// TwinCAT 3 PLC project Plc1
// ProgramVersion: 3.1.4023.0
// libraries:
//   Tc2_Standard, * (Beckhoff Automation GmbH)
//   Tc2_System, * (Beckhoff Automation GmbH)
//   Tc3_Module, * (Beckhoff Automation GmbH)
//   TcoCore, 0.9.0.4 (Vortex.Library)
//   TcoIo, 0.9.0.4 (Vortex.Library)
// project tree:
//   / PlcTask.TcTTO
//   POUs/ MAIN.TcPOU
//   DUTs/IO/PdoEntries/ Status_3D84275F.TcDUT, Ctrl_1EFB4D3B.TcDUT, Ctrl_71604E86.TcDUT, Status_B0753356.TcDUT, Status_F2CE6D91.TcDUT, U1_Status_DC903920.TcDUT, U1_Samples_25492287.TcDUT, I1_Status_DC903920.TcDUT, I1_Samples_25492287.TcDUT, U2_Status_DC903920.TcDUT, U2_Samples_25492287.TcDUT, I2_Status_DC903920.TcDUT, I2_Samples_25492287.TcDUT, U3_Status_DC903920.TcDUT, U3_Samples_25492287.TcDUT, I3_Status_DC903920.TcDUT, I3_Samples_25492287.TcDUT, StartTimeNextLatch_02E0C1C8.TcDUT, Status_642C2ED1.TcDUT, Ctrl_77460BD3.TcDUT, Outputs_A910484D.TcDUT
//   DUTs/IO/PDOs/ COM_TxPDO_Map_Inputs_Channel_3801C95E.TcDUT, COM_RxPDO_Map_Outputs_Channel_EADA2E0D.TcDUT, Channel_830843C1.TcDUT, Channel_42CA91F7.TcDUT, AO_Output_Channel_BA7EBB7C.TcDUT, COM_Inputs_3801C95E.TcDUT, COM_Outputs_DEF408EC.TcDUT, AI_Standard_Channel_A8DF64E3.TcDUT, AI_Standard_Channel_4A394481.TcDUT, L1_Voltage_Status_7371B043.TcDUT, L1_Voltage_Samples_41AEB7FF.TcDUT, L1_Current_Status_82DECBF6.TcDUT, L1_Current_Samples_9EC08B3E.TcDUT, L2_Voltage_Status_0D1813FE.TcDUT, L2_Voltage_Samples_75D833AF.TcDUT, L2_Current_Status_FCB7684B.TcDUT, L2_Current_Samples_AAB60F6E.TcDUT, L3_Voltage_Status_273F7295.TcDUT, L3_Voltage_Samples_660A4F9F.TcDUT, L3_Current_Status_D6900920.TcDUT, L3_Current_Samples_B964735E.TcDUT, AI_NextSync1Time_6DC4D296.TcDUT, AI_Sample_Count_EA88CAD9.TcDUT, InfoData_B84DBEC5.TcDUT, MTO_Inputs_Channel_53C09E8B.TcDUT, MTO_Outputs_10x_Channel_A3C0C022.TcDUT, PM_Inputs_Channel_2F868086.TcDUT, PM_Status_data_2A9514CB.TcDUT, PM_Outputs_Channel_E5FBDE30.TcDUT, AT_x_4EC2E768.TcDUT, MDT_864618EC.TcDUT, InfoData_F60A43AC.TcDUT
//   DUTs/IO/Boxes/ EK1200_013D0B49.TcDUT, EL6002_CD897635.TcDUT, EL1809_32157CFD.TcDUT, EL2809_2B6483BD.TcDUT, EL4004_E203F875.TcDUT, EL6001_0DE01E7E.TcDUT, EL9011_D65D3D32.TcDUT, EK1100_1FC0878B.TcDUT, EK1122_1FC0878B.TcDUT, EL3174_B71BFF42.TcDUT, EL3011_7A495228.TcDUT, EL2008_E2806B95.TcDUT, EK1110_1FC0878B.TcDUT, EL1819_32157CFD.TcDUT, EL2788_E2806B95.TcDUT, EL3773_F128CC82.TcDUT, EL2258_E3B260FA.TcDUT, EL3164_B71BFF42.TcDUT, EL1008_78E8D3DD.TcDUT, EL3403_812980A6.TcDUT, EL3024_C6E76B5A.TcDUT, AX5101_1BD22F51.TcDUT
//   DUTs/IO/Devices/ SyncUnitTasks_4BE01469.TcDUT, SyncUnits_67D36DDA.TcDUT, SyncUnits_91A42BBF.TcDUT
//   DUTs/IO/Topology/ Term_1_EK1200_B38DC9A8.TcDUT, Device_1_EtherCAT_B557D6C6.TcDUT, Term_11_EK1100_B6553301.TcDUT, Term_18_EK1100_20659A8D.TcDUT, Term_25_EK1100_08217EB4.TcDUT, Term_28_EK1100_415F4A7E.TcDUT, Term_24_EK1122_39E7B5CB.TcDUT, Term_23_EK1100_C1096874.TcDUT, Term_42_EK1100_1039F2C4.TcDUT, Term_10_EK1122_152EB6C2.TcDUT, Term_9_EK1100_0DC40061.TcDUT, Device_2_EtherCAT_CA128DDC.TcDUT, Term_157_EK1100_7C4BDD77.TcDUT, Term_158_EK1100_E3D699B1.TcDUT, Term_154_EK1122_E57516AE.TcDUT, Term_153_EK1100_91C0BB48.TcDUT, Term_180_EK1100_796B7783.TcDUT, Term_182_EK1100_E6B2C35E.TcDUT, Term_179_EK1122_2A33725A.TcDUT, Term_178_EK1100_9B7E9852.TcDUT, Term_147_EK1122_CA6A5D16.TcDUT, Term_189_EK1100_06A16014.TcDUT, Term_194_EK1100_D4E2C05F.TcDUT, Term_188_EK1122_78D8AA43.TcDUT, Term_187_EK1100_648C31BD.TcDUT, Term_231_EK1100_6FCE8CEB.TcDUT, Term_233_EK1100_CB654C3B.TcDUT, Term_230_EK1122_16418046.TcDUT, Term_207_EK1100_2D36550A.TcDUT, Term_186_EK1122_75C79D52.TcDUT, Term_237_EK1122_86A8F7BD.TcDUT, Term_289_EK1100_9C677E50.TcDUT, Term_294_EK1100_DFE2A59E.TcDUT, Term_331_EK1100_B9C4E092.TcDUT, Term_333_EK1100_1D6F2042.TcDUT, Term_330_EK1122_0EDE60FE.TcDUT, Term_307_EK1100_EB8FAA41.TcDUT, Term_288_EK1122_18F8921F.TcDUT, Term_146_EK1100_439F5464.TcDUT, Device_3_EtherCAT_CA191EDE.TcDUT
//   GVLs/ GVL_iXlinker.TcGVL
// real-time tasks:
//   TASK PlcTask: cycle T#10ms, priority 20, ADS port 350
// I/O:
//   DEVICE Device 1 (EtherCAT) (disabled), AmsNetId 172.20.10.110.2.1
//     Term 1 (EK1200) [EK1200-5000 EtherCAT Power supply (2A E-Bus)]
//       Term 2 (EL6002) [EL6002 Interface 2Ch. (RS232)]
//       Term 3 (EL1809) [EL1809 16Ch. Dig. Input 24V, 3ms]
//       Term 4 (EL2809) [EL2809 16Ch. Dig. Output 24V, 0.5A]
//       Term 5 (EL4004) [EL4004 4Ch. Ana. Output 0-10V, 12bit]
//       Term 6 (EL2809) [EL2809 16Ch. Dig. Output 24V, 0.5A]
//       Term 7 (EL6001) [EL6001 Interface (RS232)]
//       Term 8 (EL9011) [EL9011 End Terminal]
//   DEVICE Device 2 (EtherCAT) (disabled), AmsNetId 172.20.10.110.3.1
//     Term 9 (EK1100) [EK1100 EtherCAT Coupler (2A E-Bus)]
//       Term 10 (EK1122) [EK1122 2 port EtherCAT junction]
//         Term 11 (EK1100) [EK1100 EtherCAT Coupler (2A E-Bus)]
//           Term 12 (EL3174-0002) [EL3174-0002 4Ch. Ana. Input +/-10V, +/-20mA 16 Bit, Isolated Channels]
//           Term 13 (EL6001) [EL6001 Interface (RS232)]
//           Term 14 (EL3011) [EL3011 4Ch. Ana. Input 0-20mA DIFF]
//           Term 15 (EL2008) [EL2008 8Ch. Dig. Output 24V, 0.5A]
//           Term 16 (EL2008) [EL2008 8Ch. Dig. Output 24V, 0.5A]
//           Term 17 (EK1110) [EK1110 EtherCAT extension]
//         Term 18 (EK1100) [EK1100 EtherCAT Coupler (2A E-Bus)]
//           Term 19 (EL1809) [EL1809 16Ch. Dig. Input 24V, 3ms]
//           Term 20 (EL2809) [EL2809 16Ch. Dig. Output 24V, 0.5A]
//           Term 21 (EL1809) [EL1809 16Ch. Dig. Input 24V, 3ms]
//           Term 22 (EL3011) [EL3011 4Ch. Ana. Input 0-20mA DIFF]
//           Term 29 (EL9011) [EL9011 End Terminal]
//         Term 23 (EK1100) [EK1100 EtherCAT Coupler (2A E-Bus)]
//           Term 24 (EK1122) [EK1122 2 port EtherCAT junction]
//             Term 25 (EK1100) [EK1100 EtherCAT Coupler (2A E-Bus)]
//               Term 26 (EL1819) [EL1819 16Ch. Dig. Input 24V, 10Ã‚Âµs]
//               Term 27 (EL1819) [EL1819 16Ch. Dig. Input 24V, 10Ã‚Âµs]
//               Term 30 (EL9011) [EL9011 End Terminal]
//             Term 28 (EK1100) [EK1100 EtherCAT Coupler (2A E-Bus)]
//               Term 29 (EL2788) [EL2788 8Ch. Dig. Output 24V AC/DC, 2A]
//               Term 30 (EL3773) [EL3773 3 Ch. Power Monitoring, Oversample]
//               Term 31 (EL9011) [EL9011 End Terminal]
//           Term 31 (EL3773) [EL3773 3 Ch. Power Monitoring, Oversample]
//           Term 32 (EL2258) [EL2258 8Ch. Dig Output 24V with Multi-Time-Stamp]
//           Term 33 (EL3164) [EL3164 4Ch. Ana. Input 0-10V]
//           Term 40 (EK1110) [EK1110 EtherCAT extension]
//         Term 42 (EK1100) [EK1100 EtherCAT Coupler (2A E-Bus)]
//           Term 43 (EL1008) [EL1008 8Ch. Dig. Input 24V, 3ms]
//           Term 44 (EL1008) [EL1008 8Ch. Dig. Input 24V, 3ms]
//       Term 34 (EL3403) [EL3403 3Ch. Power Measuring]
//       Term 35 (EL6001) [EL6001 Interface (RS232)]
//       Term 36 (EL3024) [EL3024 4Ch. Ana. Input 4-20mA DIFF]
//       Term 33 (EL9011) [EL9011 End Terminal]
//   DEVICE Device 3 (EtherCAT) (disabled), AmsNetId 172.20.10.110.4.1
//     Term 146 (EK1100) [EK1100 EtherCAT Coupler (2A E-Bus)]
//       Term 147 (EK1122) [EK1122 2 port EtherCAT junction]
//         Term 153 (EK1100) [EK1100 EtherCAT Coupler (2A E-Bus)]
//           Term 154 (EK1122) [EK1122 2 port EtherCAT junction]
//             Term 157 (EK1100) [EK1100 EtherCAT Coupler (2A E-Bus)]
//               Term 159 (EL1809) [EL1809 16Ch. Dig. Input 24V, 3ms]
//             Term 158 (EK1100) [EK1100 EtherCAT Coupler (2A E-Bus)]
//               Term 160 (EL1809) [EL1809 16Ch. Dig. Input 24V, 3ms]
//           Term 155 (EL2008) [EL2008 8Ch. Dig. Output 24V, 0.5A]
//           Term 156 (EL2008) [EL2008 8Ch. Dig. Output 24V, 0.5A]
//         Term 178 (EK1100) [EK1100 EtherCAT Coupler (2A E-Bus)]
//           Term 179 (EK1122) [EK1122 2 port EtherCAT junction]
//             Term 180 (EK1100) [EK1100 EtherCAT Coupler (2A E-Bus)]
//               Term 181 (EL1809) [EL1809 16Ch. Dig. Input 24V, 3ms]
//             Term 182 (EK1100) [EK1100 EtherCAT Coupler (2A E-Bus)]
//               Term 183 (EL1809) [EL1809 16Ch. Dig. Input 24V, 3ms]
//           Term 184 (EL2008) [EL2008 8Ch. Dig. Output 24V, 0.5A]
//           Term 185 (EL2008) [EL2008 8Ch. Dig. Output 24V, 0.5A]
//       Term 186 (EK1122) [EK1122 2 port EtherCAT junction]
//         Term 187 (EK1100) [EK1100 EtherCAT Coupler (2A E-Bus)]
//           Term 188 (EK1122) [EK1122 2 port EtherCAT junction]
//             Term 189 (EK1100) [EK1100 EtherCAT Coupler (2A E-Bus)]
//               Term 193 (EL1809) [EL1809 16Ch. Dig. Input 24V, 3ms]
//             Term 194 (EK1100) [EK1100 EtherCAT Coupler (2A E-Bus)]
//               Term 200 (EL1809) [EL1809 16Ch. Dig. Input 24V, 3ms]
//           Term 204 (EL2008) [EL2008 8Ch. Dig. Output 24V, 0.5A]
//           Term 205 (EL2008) [EL2008 8Ch. Dig. Output 24V, 0.5A]
//         Term 207 (EK1100) [EK1100 EtherCAT Coupler (2A E-Bus)]
//           Term 230 (EK1122) [EK1122 2 port EtherCAT junction]
//             Term 231 (EK1100) [EK1100 EtherCAT Coupler (2A E-Bus)]
//               Term 232 (EL1809) [EL1809 16Ch. Dig. Input 24V, 3ms]
//             Term 233 (EK1100) [EK1100 EtherCAT Coupler (2A E-Bus)]
//               Term 234 (EL1809) [EL1809 16Ch. Dig. Input 24V, 3ms]
//           Term 235 (EL2008) [EL2008 8Ch. Dig. Output 24V, 0.5A]
//           Term 236 (EL2008) [EL2008 8Ch. Dig. Output 24V, 0.5A]
//       Term 148 (EL1809) [EL1809 16Ch. Dig. Input 24V, 3ms]
//       Term 149 (EL1809) [EL1809 16Ch. Dig. Input 24V, 3ms]
//       Term 150 (EL1809) [EL1809 16Ch. Dig. Input 24V, 3ms]
//       Term 151 (EL1809) [EL1809 16Ch. Dig. Input 24V, 3ms]
//       Term 152 (EL1809) [EL1809 16Ch. Dig. Input 24V, 3ms]
//       Term 288 (EK1122) [EK1122 2 port EtherCAT junction]
//         Term 289 (EK1100) [EK1100 EtherCAT Coupler (2A E-Bus)]
//           Term 237 (EK1122) [EK1122 2 port EtherCAT junction]
//             Drive 238 (AX5101-0000-0214) [AX5101-0000-0214 EtherCAT Drive (SoE, 1 Ch.)]
//           Term 293 (EL1809) [EL1809 16Ch. Dig. Input 24V, 3ms]
//         Term 294 (EK1100) [EK1100 EtherCAT Coupler (2A E-Bus)]
//           Term 300 (EL1809) [EL1809 16Ch. Dig. Input 24V, 3ms]
//           Term 304 (EL2008) [EL2008 8Ch. Dig. Output 24V, 0.5A]
//           Term 305 (EL2008) [EL2008 8Ch. Dig. Output 24V, 0.5A]
//         Term 307 (EK1100) [EK1100 EtherCAT Coupler (2A E-Bus)]
//           Term 330 (EK1122) [EK1122 2 port EtherCAT junction]
//             Term 331 (EK1100) [EK1100 EtherCAT Coupler (2A E-Bus)]
//               Term 332 (EL1809) [EL1809 16Ch. Dig. Input 24V, 3ms]
//             Term 333 (EK1100) [EK1100 EtherCAT Coupler (2A E-Bus)]
//               Term 334 (EL1809) [EL1809 16Ch. Dig. Input 24V, 3ms]
//           Term 335 (EL2008) [EL2008 8Ch. Dig. Output 24V, 0.5A]
//           Term 336 (EL2008) [EL2008 8Ch. Dig. Output 24V, 0.5A]
//       Term 1158 (EL2008) [EL2008 8Ch. Dig. Output 24V, 0.5A]
//       Term 1159 (EL2008) [EL2008 8Ch. Dig. Output 24V, 0.5A]
//       Term 1160 (EL2008) [EL2008 8Ch. Dig. Output 24V, 0.5A]
//       Term 1161 (EL2008) [EL2008 8Ch. Dig. Output 24V, 0.5A]
//       Term 1162 (EL2008) [EL2008 8Ch. Dig. Output 24V, 0.5A]
//       Term 1163 (EL2008) [EL2008 8Ch. Dig. Output 24V, 0.5A]
// variable links:
//   Plc1/Plc1 Instance <-> Device 1 (EtherCAT)
//     PlcTask Inputs/GVL_iXlinker.Device_1_EtherCAT.InfoData.AmsNetId <-> InfoData/AmsNetId
//     PlcTask Inputs/GVL_iXlinker.Device_1_EtherCAT.InfoData.CfgSlaveCount <-> InfoData/CfgSlaveCount
//     PlcTask Inputs/GVL_iXlinker.Device_1_EtherCAT.InfoData.ChangeCount <-> InfoData/ChangeCount
//     PlcTask Inputs/GVL_iXlinker.Device_1_EtherCAT.InfoData.DcToExtTimeOffset <-> InfoData/DcToExtTimeOffset
//     PlcTask Inputs/GVL_iXlinker.Device_1_EtherCAT.InfoData.DcToTcTimeOffset <-> InfoData/DcToTcTimeOffset
//     PlcTask Inputs/GVL_iXlinker.Device_1_EtherCAT.InfoData.DevId <-> InfoData/DevId
//     PlcTask Inputs/GVL_iXlinker.Device_1_EtherCAT.Inputs.DevState <-> Inputs/DevState
//     PlcTask Inputs/GVL_iXlinker.Device_1_EtherCAT.Inputs.Frm0InputToggle <-> Inputs/Frm0InputToggle
//     PlcTask Inputs/GVL_iXlinker.Device_1_EtherCAT.Inputs.Frm0State <-> Inputs/Frm0State
//     PlcTask Inputs/GVL_iXlinker.Device_1_EtherCAT.Inputs.Frm0WcState <-> Inputs/Frm0WcState
//     PlcTask Inputs/GVL_iXlinker.Device_1_EtherCAT.Inputs.SlaveCount <-> Inputs/SlaveCount
//     PlcTask Inputs/GVL_iXlinker.Device_1_EtherCAT.SyncUnits._default.PlcTask.InfoData.ObjectId <-> SyncUnits/<default>/PlcTask/InfoData/ObjectId
//     PlcTask Inputs/GVL_iXlinker.Device_1_EtherCAT.SyncUnits._default.PlcTask.InfoData.SlaveCount <-> SyncUnits/<default>/PlcTask/InfoData/SlaveCount
//     PlcTask Inputs/GVL_iXlinker.Device_1_EtherCAT.SyncUnits._default.PlcTask.InfoData.State <-> SyncUnits/<default>/PlcTask/InfoData/State
//     PlcTask Inputs/GVL_iXlinker.Device_1_EtherCAT.SyncUnits._default.PlcTask.WcState.WcState <-> SyncUnits/<default>/PlcTask/WcState/WcState
//     PlcTask Outputs/GVL_iXlinker.Device_1_EtherCAT.Outputs.DevCtrl <-> Outputs/DevCtrl
//     PlcTask Outputs/GVL_iXlinker.Device_1_EtherCAT.Outputs.Frm0Ctrl <-> Outputs/Frm0Ctrl
//     PlcTask Outputs/GVL_iXlinker.Device_1_EtherCAT.Outputs.Frm0WcCtrl <-> Outputs/Frm0WcCtrl
//   Plc1/Plc1 Instance <-> Device 1 (EtherCAT)/Term 1 (EK1200)/Term 2 (EL6002)
//     PlcTask Inputs/GVL_iXlinker.Device_1_EtherCAT.Term_1_EK1200.Term_2_EL6002.COM_TxPDO_Map_Inputs_Channel_1.Data_In[0] <-> COM TxPDO-Map Inputs Channel 1/Data In 0
//     PlcTask Inputs/GVL_iXlinker.Device_1_EtherCAT.Term_1_EK1200.Term_2_EL6002.COM_TxPDO_Map_Inputs_Channel_1.Data_In[10] <-> COM TxPDO-Map Inputs Channel 1/Data In 10
//     PlcTask Inputs/GVL_iXlinker.Device_1_EtherCAT.Term_1_EK1200.Term_2_EL6002.COM_TxPDO_Map_Inputs_Channel_1.Data_In[11] <-> COM TxPDO-Map Inputs Channel 1/Data In 11
//     PlcTask Inputs/GVL_iXlinker.Device_1_EtherCAT.Term_1_EK1200.Term_2_EL6002.COM_TxPDO_Map_Inputs_Channel_1.Data_In[12] <-> COM TxPDO-Map Inputs Channel 1/Data In 12
//     PlcTask Inputs/GVL_iXlinker.Device_1_EtherCAT.Term_1_EK1200.Term_2_EL6002.COM_TxPDO_Map_Inputs_Channel_1.Data_In[13] <-> COM TxPDO-Map Inputs Channel 1/Data In 13
//     PlcTask Inputs/GVL_iXlinker.Device_1_EtherCAT.Term_1_EK1200.Term_2_EL6002.COM_TxPDO_Map_Inputs_Channel_1.Data_In[14] <-> COM TxPDO-Map Inputs Channel 1/Data In 14
//     PlcTask Inputs/GVL_iXlinker.Device_1_EtherCAT.Term_1_EK1200.Term_2_EL6002.COM_TxPDO_Map_Inputs_Channel_1.Data_In[15] <-> COM TxPDO-Map Inputs Channel 1/Data In 15
//     PlcTask Inputs/GVL_iXlinker.Device_1_EtherCAT.Term_1_EK1200.Term_2_EL6002.COM_TxPDO_Map_Inputs_Channel_1.Data_In[16] <-> COM TxPDO-Map Inputs Channel 1/Data In 16
//     PlcTask Inputs/GVL_iXlinker.Device_1_EtherCAT.Term_1_EK1200.Term_2_EL6002.COM_TxPDO_Map_Inputs_Channel_1.Data_In[17] <-> COM TxPDO-Map Inputs Channel 1/Data In 17
//     PlcTask Inputs/GVL_iXlinker.Device_1_EtherCAT.Term_1_EK1200.Term_2_EL6002.COM_TxPDO_Map_Inputs_Channel_1.Data_In[18] <-> COM TxPDO-Map Inputs Channel 1/Data In 18
//     PlcTask Inputs/GVL_iXlinker.Device_1_EtherCAT.Term_1_EK1200.Term_2_EL6002.COM_TxPDO_Map_Inputs_Channel_1.Data_In[19] <-> COM TxPDO-Map Inputs Channel 1/Data In 19
//     PlcTask Inputs/GVL_iXlinker.Device_1_EtherCAT.Term_1_EK1200.Term_2_EL6002.COM_TxPDO_Map_Inputs_Channel_1.Data_In[1] <-> COM TxPDO-Map Inputs Channel 1/Data In 1
//     PlcTask Inputs/GVL_iXlinker.Device_1_EtherCAT.Term_1_EK1200.Term_2_EL6002.COM_TxPDO_Map_Inputs_Channel_1.Data_In[20] <-> COM TxPDO-Map Inputs Channel 1/Data In 20
//     PlcTask Inputs/GVL_iXlinker.Device_1_EtherCAT.Term_1_EK1200.Term_2_EL6002.COM_TxPDO_Map_Inputs_Channel_1.Data_In[21] <-> COM TxPDO-Map Inputs Channel 1/Data In 21
//     PlcTask Inputs/GVL_iXlinker.Device_1_EtherCAT.Term_1_EK1200.Term_2_EL6002.COM_TxPDO_Map_Inputs_Channel_1.Data_In[2] <-> COM TxPDO-Map Inputs Channel 1/Data In 2
//     PlcTask Inputs/GVL_iXlinker.Device_1_EtherCAT.Term_1_EK1200.Term_2_EL6002.COM_TxPDO_Map_Inputs_Channel_1.Data_In[3] <-> COM TxPDO-Map Inputs Channel 1/Data In 3
//     PlcTask Inputs/GVL_iXlinker.Device_1_EtherCAT.Term_1_EK1200.Term_2_EL6002.COM_TxPDO_Map_Inputs_Channel_1.Data_In[4] <-> COM TxPDO-Map Inputs Channel 1/Data In 4
//     PlcTask Inputs/GVL_iXlinker.Device_1_EtherCAT.Term_1_EK1200.Term_2_EL6002.COM_TxPDO_Map_Inputs_Channel_1.Data_In[5] <-> COM TxPDO-Map Inputs Channel 1/Data In 5
//     PlcTask Inputs/GVL_iXlinker.Device_1_EtherCAT.Term_1_EK1200.Term_2_EL6002.COM_TxPDO_Map_Inputs_Channel_1.Data_In[6] <-> COM TxPDO-Map Inputs Channel 1/Data In 6
//     PlcTask Inputs/GVL_iXlinker.Device_1_EtherCAT.Term_1_EK1200.Term_2_EL6002.COM_TxPDO_Map_Inputs_Channel_1.Data_In[7] <-> COM TxPDO-Map Inputs Channel 1/Data In 7
//     PlcTask Inputs/GVL_iXlinker.Device_1_EtherCAT.Term_1_EK1200.Term_2_EL6002.COM_TxPDO_Map_Inputs_Channel_1.Data_In[8] <-> COM TxPDO-Map Inputs Channel 1/Data In 8
//     PlcTask Inputs/GVL_iXlinker.Device_1_EtherCAT.Term_1_EK1200.Term_2_EL6002.COM_TxPDO_Map_Inputs_Channel_1.Data_In[9] <-> COM TxPDO-Map Inputs Channel 1/Data In 9
//     PlcTask Inputs/GVL_iXlinker.Device_1_EtherCAT.Term_1_EK1200.Term_2_EL6002.COM_TxPDO_Map_Inputs_Channel_2.Data_In[0] <-> COM TxPDO-Map Inputs Channel 2/Data In 0
//     PlcTask Inputs/GVL_iXlinker.Device_1_EtherCAT.Term_1_EK1200.Term_2_EL6002.COM_TxPDO_Map_Inputs_Channel_2.Data_In[10] <-> COM TxPDO-Map Inputs Channel 2/Data In 10
//     PlcTask Inputs/GVL_iXlinker.Device_1_EtherCAT.Term_1_EK1200.Term_2_EL6002.COM_TxPDO_Map_Inputs_Channel_2.Data_In[11] <-> COM TxPDO-Map Inputs Channel 2/Data In 11
//     PlcTask Inputs/GVL_iXlinker.Device_1_EtherCAT.Term_1_EK1200.Term_2_EL6002.COM_TxPDO_Map_Inputs_Channel_2.Data_In[12] <-> COM TxPDO-Map Inputs Channel 2/Data In 12
//     PlcTask Inputs/GVL_iXlinker.Device_1_EtherCAT.Term_1_EK1200.Term_2_EL6002.COM_TxPDO_Map_Inputs_Channel_2.Data_In[13] <-> COM TxPDO-Map Inputs Channel 2/Data In 13
//     PlcTask Inputs/GVL_iXlinker.Device_1_EtherCAT.Term_1_EK1200.Term_2_EL6002.COM_TxPDO_Map_Inputs_Channel_2.Data_In[14] <-> COM TxPDO-Map Inputs Channel 2/Data In 14
//     PlcTask Inputs/GVL_iXlinker.Device_1_EtherCAT.Term_1_EK1200.Term_2_EL6002.COM_TxPDO_Map_Inputs_Channel_2.Data_In[15] <-> COM TxPDO-Map Inputs Channel 2/Data In 15
//     PlcTask Inputs/GVL_iXlinker.Device_1_EtherCAT.Term_1_EK1200.Term_2_EL6002.COM_TxPDO_Map_Inputs_Channel_2.Data_In[16] <-> COM TxPDO-Map Inputs Channel 2/Data In 16
//     PlcTask Inputs/GVL_iXlinker.Device_1_EtherCAT.Term_1_EK1200.Term_2_EL6002.COM_TxPDO_Map_Inputs_Channel_2.Data_In[17] <-> COM TxPDO-Map Inputs Channel 2/Data In 17
//     PlcTask Inputs/GVL_iXlinker.Device_1_EtherCAT.Term_1_EK1200.Term_2_EL6002.COM_TxPDO_Map_Inputs_Channel_2.Data_In[18] <-> COM TxPDO-Map Inputs Channel 2/Data In 18
//     PlcTask Inputs/GVL_iXlinker.Device_1_EtherCAT.Term_1_EK1200.Term_2_EL6002.COM_TxPDO_Map_Inputs_Channel_2.Data_In[19] <-> COM TxPDO-Map Inputs Channel 2/Data In 19
//     PlcTask Inputs/GVL_iXlinker.Device_1_EtherCAT.Term_1_EK1200.Term_2_EL6002.COM_TxPDO_Map_Inputs_Channel_2.Data_In[1] <-> COM TxPDO-Map Inputs Channel 2/Data In 1
//     PlcTask Inputs/GVL_iXlinker.Device_1_EtherCAT.Term_1_EK1200.Term_2_EL6002.COM_TxPDO_Map_Inputs_Channel_2.Data_In[20] <-> COM TxPDO-Map Inputs Channel 2/Data In 20
//     PlcTask Inputs/GVL_iXlinker.Device_1_EtherCAT.Term_1_EK1200.Term_2_EL6002.COM_TxPDO_Map_Inputs_Channel_2.Data_In[21] <-> COM TxPDO-Map Inputs Channel 2/Data In 21
//     PlcTask Inputs/GVL_iXlinker.Device_1_EtherCAT.Term_1_EK1200.Term_2_EL6002.COM_TxPDO_Map_Inputs_Channel_2.Data_In[2] <-> COM TxPDO-Map Inputs Channel 2/Data In 2
//     PlcTask Inputs/GVL_iXlinker.Device_1_EtherCAT.Term_1_EK1200.Term_2_EL6002.COM_TxPDO_Map_Inputs_Channel_2.Data_In[3] <-> COM TxPDO-Map Inputs Channel 2/Data In 3
//     PlcTask Inputs/GVL_iXlinker.Device_1_EtherCAT.Term_1_EK1200.Term_2_EL6002.COM_TxPDO_Map_Inputs_Channel_2.Data_In[4] <-> COM TxPDO-Map Inputs Channel 2/Data In 4
//     PlcTask Inputs/GVL_iXlinker.Device_1_EtherCAT.Term_1_EK1200.Term_2_EL6002.COM_TxPDO_Map_Inputs_Channel_2.Data_In[5] <-> COM TxPDO-Map Inputs Channel 2/Data In 5
//     PlcTask Inputs/GVL_iXlinker.Device_1_EtherCAT.Term_1_EK1200.Term_2_EL6002.COM_TxPDO_Map_Inputs_Channel_2.Data_In[6] <-> COM TxPDO-Map Inputs Channel 2/Data In 6
//     PlcTask Inputs/GVL_iXlinker.Device_1_EtherCAT.Term_1_EK1200.Term_2_EL6002.COM_TxPDO_Map_Inputs_Channel_2.Data_In[7] <-> COM TxPDO-Map Inputs Channel 2/Data In 7
//     PlcTask Inputs/GVL_iXlinker.Device_1_EtherCAT.Term_1_EK1200.Term_2_EL6002.COM_TxPDO_Map_Inputs_Channel_2.Data_In[8] <-> COM TxPDO-Map Inputs Channel 2/Data In 8
//     PlcTask Inputs/GVL_iXlinker.Device_1_EtherCAT.Term_1_EK1200.Term_2_EL6002.COM_TxPDO_Map_Inputs_Channel_2.Data_In[9] <-> COM TxPDO-Map Inputs Channel 2/Data In 9
//     PlcTask Inputs/GVL_iXlinker.Device_1_EtherCAT.Term_1_EK1200.Term_2_EL6002.COM_TxPDO_Map_Inputs_Channel_1.Status/Buffer_full <-> COM TxPDO-Map Inputs Channel 1/Status/Buffer full
//     PlcTask Inputs/GVL_iXlinker.Device_1_EtherCAT.Term_1_EK1200.Term_2_EL6002.COM_TxPDO_Map_Inputs_Channel_2.Status/Buffer_full <-> COM TxPDO-Map Inputs Channel 2/Status/Buffer full
//     PlcTask Inputs/GVL_iXlinker.Device_1_EtherCAT.Term_1_EK1200.Term_2_EL6002.COM_TxPDO_Map_Inputs_Channel_1.Status/Framing_error <-> COM TxPDO-Map Inputs Channel 1/Status/Framing error
//     PlcTask Inputs/GVL_iXlinker.Device_1_EtherCAT.Term_1_EK1200.Term_2_EL6002.COM_TxPDO_Map_Inputs_Channel_2.Status/Framing_error <-> COM TxPDO-Map Inputs Channel 2/Status/Framing error
//     PlcTask Inputs/GVL_iXlinker.Device_1_EtherCAT.Term_1_EK1200.Term_2_EL6002.COM_TxPDO_Map_Inputs_Channel_1.Status/Init_accepted <-> COM TxPDO-Map Inputs Channel 1/Status/Init accepted
//     PlcTask Inputs/GVL_iXlinker.Device_1_EtherCAT.Term_1_EK1200.Term_2_EL6002.COM_TxPDO_Map_Inputs_Channel_2.Status/Init_accepted <-> COM TxPDO-Map Inputs Channel 2/Status/Init accepted
//     PlcTask Inputs/GVL_iXlinker.Device_1_EtherCAT.Term_1_EK1200.Term_2_EL6002.COM_TxPDO_Map_Inputs_Channel_1.Status/Input_length <-> COM TxPDO-Map Inputs Channel 1/Status/Input length
//     PlcTask Inputs/GVL_iXlinker.Device_1_EtherCAT.Term_1_EK1200.Term_2_EL6002.COM_TxPDO_Map_Inputs_Channel_2.Status/Input_length <-> COM TxPDO-Map Inputs Channel 2/Status/Input length
//     PlcTask Inputs/GVL_iXlinker.Device_1_EtherCAT.Term_1_EK1200.Term_2_EL6002.COM_TxPDO_Map_Inputs_Channel_1.Status/Overrun_error <-> COM TxPDO-Map Inputs Channel 1/Status/Overrun error
//     PlcTask Inputs/GVL_iXlinker.Device_1_EtherCAT.Term_1_EK1200.Term_2_EL6002.COM_TxPDO_Map_Inputs_Channel_2.Status/Overrun_error <-> COM TxPDO-Map Inputs Channel 2/Status/Overrun error
//     PlcTask Inputs/GVL_iXlinker.Device_1_EtherCAT.Term_1_EK1200.Term_2_EL6002.COM_TxPDO_Map_Inputs_Channel_1.Status/Parity_error <-> COM TxPDO-Map Inputs Channel 1/Status/Parity error
//     PlcTask Inputs/GVL_iXlinker.Device_1_EtherCAT.Term_1_EK1200.Term_2_EL6002.COM_TxPDO_Map_Inputs_Channel_2.Status/Parity_error <-> COM TxPDO-Map Inputs Channel 2/Status/Parity error
//     PlcTask Inputs/GVL_iXlinker.Device_1_EtherCAT.Term_1_EK1200.Term_2_EL6002.COM_TxPDO_Map_Inputs_Channel_1.Status/Receive_request <-> COM TxPDO-Map Inputs Channel 1/Status/Receive request
//     PlcTask Inputs/GVL_iXlinker.Device_1_EtherCAT.Term_1_EK1200.Term_2_EL6002.COM_TxPDO_Map_Inputs_Channel_2.Status/Receive_request <-> COM TxPDO-Map Inputs Channel 2/Status/Receive request
//     PlcTask Inputs/GVL_iXlinker.Device_1_EtherCAT.Term_1_EK1200.Term_2_EL6002.COM_TxPDO_Map_Inputs_Channel_1.Status/Transmit_accepted <-> COM TxPDO-Map Inputs Channel 1/Status/Transmit accepted
//     PlcTask Inputs/GVL_iXlinker.Device_1_EtherCAT.Term_1_EK1200.Term_2_EL6002.COM_TxPDO_Map_Inputs_Channel_2.Status/Transmit_accepted <-> COM TxPDO-Map Inputs Channel 2/Status/Transmit accepted
//     PlcTask Inputs/GVL_iXlinker.Device_1_EtherCAT.Term_1_EK1200.Term_2_EL6002.InfoData.AdsAddr <-> InfoData/AdsAddr
//     PlcTask Inputs/GVL_iXlinker.Device_1_EtherCAT.Term_1_EK1200.Term_2_EL6002.InfoData.State <-> InfoData/State
//     PlcTask Inputs/GVL_iXlinker.Device_1_EtherCAT.Term_1_EK1200.Term_2_EL6002.WcState.InputToggle <-> WcState/InputToggle
//     PlcTask Inputs/GVL_iXlinker.Device_1_EtherCAT.Term_1_EK1200.Term_2_EL6002.WcState.WcState <-> WcState/WcState
//     PlcTask Outputs/GVL_iXlinker.Device_1_EtherCAT.Term_1_EK1200.Term_2_EL6002.COM_RxPDO_Map_Outputs_Channel_1.Ctrl/Init_request <-> COM RxPDO-Map Outputs Channel 1/Ctrl/Init request
//     PlcTask Outputs/GVL_iXlinker.Device_1_EtherCAT.Term_1_EK1200.Term_2_EL6002.COM_RxPDO_Map_Outputs_Channel_2.Ctrl/Init_request <-> COM RxPDO-Map Outputs Channel 2/Ctrl/Init request
//     PlcTask Outputs/GVL_iXlinker.Device_1_EtherCAT.Term_1_EK1200.Term_2_EL6002.COM_RxPDO_Map_Outputs_Channel_1.Ctrl/Output_length <-> COM RxPDO-Map Outputs Channel 1/Ctrl/Output length
//     PlcTask Outputs/GVL_iXlinker.Device_1_EtherCAT.Term_1_EK1200.Term_2_EL6002.COM_RxPDO_Map_Outputs_Channel_2.Ctrl/Output_length <-> COM RxPDO-Map Outputs Channel 2/Ctrl/Output length
//     PlcTask Outputs/GVL_iXlinker.Device_1_EtherCAT.Term_1_EK1200.Term_2_EL6002.COM_RxPDO_Map_Outputs_Channel_1.Ctrl/Receive_accepted <-> COM RxPDO-Map Outputs Channel 1/Ctrl/Receive accepted
//     PlcTask Outputs/GVL_iXlinker.Device_1_EtherCAT.Term_1_EK1200.Term_2_EL6002.COM_RxPDO_Map_Outputs_Channel_2.Ctrl/Receive_accepted <-> COM RxPDO-Map Outputs Channel 2/Ctrl/Receive accepted
//     PlcTask Outputs/GVL_iXlinker.Device_1_EtherCAT.Term_1_EK1200.Term_2_EL6002.COM_RxPDO_Map_Outputs_Channel_1.Ctrl/Send_continuous <-> COM RxPDO-Map Outputs Channel 1/Ctrl/Send continuous
//     PlcTask Outputs/GVL_iXlinker.Device_1_EtherCAT.Term_1_EK1200.Term_2_EL6002.COM_RxPDO_Map_Outputs_Channel_2.Ctrl/Send_continuous <-> COM RxPDO-Map Outputs Channel 2/Ctrl/Send continuous
//     PlcTask Outputs/GVL_iXlinker.Device_1_EtherCAT.Term_1_EK1200.Term_2_EL6002.COM_RxPDO_Map_Outputs_Channel_1.Ctrl/Transmit_request <-> COM RxPDO-Map Outputs Channel 1/Ctrl/Transmit request
//     PlcTask Outputs/GVL_iXlinker.Device_1_EtherCAT.Term_1_EK1200.Term_2_EL6002.COM_RxPDO_Map_Outputs_Channel_2.Ctrl/Transmit_request <-> COM RxPDO-Map Outputs Channel 2/Ctrl/Transmit request
//     PlcTask Outputs/GVL_iXlinker.Device_1_EtherCAT.Term_1_EK1200.Term_2_EL6002.COM_RxPDO_Map_Outputs_Channel_1.Data_Out[0] <-> COM RxPDO-Map Outputs Channel 1/Data Out 0
//     PlcTask Outputs/GVL_iXlinker.Device_1_EtherCAT.Term_1_EK1200.Term_2_EL6002.COM_RxPDO_Map_Outputs_Channel_1.Data_Out[10] <-> COM RxPDO-Map Outputs Channel 1/Data Out 10
//     PlcTask Outputs/GVL_iXlinker.Device_1_EtherCAT.Term_1_EK1200.Term_2_EL6002.COM_RxPDO_Map_Outputs_Channel_1.Data_Out[11] <-> COM RxPDO-Map Outputs Channel 1/Data Out 11
//     PlcTask Outputs/GVL_iXlinker.Device_1_EtherCAT.Term_1_EK1200.Term_2_EL6002.COM_RxPDO_Map_Outputs_Channel_1.Data_Out[12] <-> COM RxPDO-Map Outputs Channel 1/Data Out 12
//     PlcTask Outputs/GVL_iXlinker.Device_1_EtherCAT.Term_1_EK1200.Term_2_EL6002.COM_RxPDO_Map_Outputs_Channel_1.Data_Out[13] <-> COM RxPDO-Map Outputs Channel 1/Data Out 13
//     PlcTask Outputs/GVL_iXlinker.Device_1_EtherCAT.Term_1_EK1200.Term_2_EL6002.COM_RxPDO_Map_Outputs_Channel_1.Data_Out[14] <-> COM RxPDO-Map Outputs Channel 1/Data Out 14
//     PlcTask Outputs/GVL_iXlinker.Device_1_EtherCAT.Term_1_EK1200.Term_2_EL6002.COM_RxPDO_Map_Outputs_Channel_1.Data_Out[15] <-> COM RxPDO-Map Outputs Channel 1/Data Out 15
//     PlcTask Outputs/GVL_iXlinker.Device_1_EtherCAT.Term_1_EK1200.Term_2_EL6002.COM_RxPDO_Map_Outputs_Channel_1.Data_Out[16] <-> COM RxPDO-Map Outputs Channel 1/Data Out 16
//     PlcTask Outputs/GVL_iXlinker.Device_1_EtherCAT.Term_1_EK1200.Term_2_EL6002.COM_RxPDO_Map_Outputs_Channel_1.Data_Out[17] <-> COM RxPDO-Map Outputs Channel 1/Data Out 17
//     PlcTask Outputs/GVL_iXlinker.Device_1_EtherCAT.Term_1_EK1200.Term_2_EL6002.COM_RxPDO_Map_Outputs_Channel_1.Data_Out[18] <-> COM RxPDO-Map Outputs Channel 1/Data Out 18
//     PlcTask Outputs/GVL_iXlinker.Device_1_EtherCAT.Term_1_EK1200.Term_2_EL6002.COM_RxPDO_Map_Outputs_Channel_1.Data_Out[19] <-> COM RxPDO-Map Outputs Channel 1/Data Out 19
//     PlcTask Outputs/GVL_iXlinker.Device_1_EtherCAT.Term_1_EK1200.Term_2_EL6002.COM_RxPDO_Map_Outputs_Channel_1.Data_Out[1] <-> COM RxPDO-Map Outputs Channel 1/Data Out 1
//     PlcTask Outputs/GVL_iXlinker.Device_1_EtherCAT.Term_1_EK1200.Term_2_EL6002.COM_RxPDO_Map_Outputs_Channel_1.Data_Out[20] <-> COM RxPDO-Map Outputs Channel 1/Data Out 20
//     PlcTask Outputs/GVL_iXlinker.Device_1_EtherCAT.Term_1_EK1200.Term_2_EL6002.COM_RxPDO_Map_Outputs_Channel_1.Data_Out[21] <-> COM RxPDO-Map Outputs Channel 1/Data Out 21
//     PlcTask Outputs/GVL_iXlinker.Device_1_EtherCAT.Term_1_EK1200.Term_2_EL6002.COM_RxPDO_Map_Outputs_Channel_1.Data_Out[2] <-> COM RxPDO-Map Outputs Channel 1/Data Out 2
//     PlcTask Outputs/GVL_iXlinker.Device_1_EtherCAT.Term_1_EK1200.Term_2_EL6002.COM_RxPDO_Map_Outputs_Channel_1.Data_Out[3] <-> COM RxPDO-Map Outputs Channel 1/Data Out 3
//     PlcTask Outputs/GVL_iXlinker.Device_1_EtherCAT.Term_1_EK1200.Term_2_EL6002.COM_RxPDO_Map_Outputs_Channel_1.Data_Out[4] <-> COM RxPDO-Map Outputs Channel 1/Data Out 4
//     PlcTask Outputs/GVL_iXlinker.Device_1_EtherCAT.Term_1_EK1200.Term_2_EL6002.COM_RxPDO_Map_Outputs_Channel_1.Data_Out[5] <-> COM RxPDO-Map Outputs Channel 1/Data Out 5
//     PlcTask Outputs/GVL_iXlinker.Device_1_EtherCAT.Term_1_EK1200.Term_2_EL6002.COM_RxPDO_Map_Outputs_Channel_1.Data_Out[6] <-> COM RxPDO-Map Outputs Channel 1/Data Out 6
//     PlcTask Outputs/GVL_iXlinker.Device_1_EtherCAT.Term_1_EK1200.Term_2_EL6002.COM_RxPDO_Map_Outputs_Channel_1.Data_Out[7] <-> COM RxPDO-Map Outputs Channel 1/Data Out 7
//     PlcTask Outputs/GVL_iXlinker.Device_1_EtherCAT.Term_1_EK1200.Term_2_EL6002.COM_RxPDO_Map_Outputs_Channel_1.Data_Out[8] <-> COM RxPDO-Map Outputs Channel 1/Data Out 8
//     PlcTask Outputs/GVL_iXlinker.Device_1_EtherCAT.Term_1_EK1200.Term_2_EL6002.COM_RxPDO_Map_Outputs_Channel_1.Data_Out[9] <-> COM RxPDO-Map Outputs Channel 1/Data Out 9
//     PlcTask Outputs/GVL_iXlinker.Device_1_EtherCAT.Term_1_EK1200.Term_2_EL6002.COM_RxPDO_Map_Outputs_Channel_2.Data_Out[0] <-> COM RxPDO-Map Outputs Channel 2/Data Out 0
//     PlcTask Outputs/GVL_iXlinker.Device_1_EtherCAT.Term_1_EK1200.Term_2_EL6002.COM_RxPDO_Map_Outputs_Channel_2.Data_Out[10] <-> COM RxPDO-Map Outputs Channel 2/Data Out 10
//     PlcTask Outputs/GVL_iXlinker.Device_1_EtherCAT.Term_1_EK1200.Term_2_EL6002.COM_RxPDO_Map_Outputs_Channel_2.Data_Out[11] <-> COM RxPDO-Map Outputs Channel 2/Data Out 11
//     PlcTask Outputs/GVL_iXlinker.Device_1_EtherCAT.Term_1_EK1200.Term_2_EL6002.COM_RxPDO_Map_Outputs_Channel_2.Data_Out[12] <-> COM RxPDO-Map Outputs Channel 2/Data Out 12
//     PlcTask Outputs/GVL_iXlinker.Device_1_EtherCAT.Term_1_EK1200.Term_2_EL6002.COM_RxPDO_Map_Outputs_Channel_2.Data_Out[13] <-> COM RxPDO-Map Outputs Channel 2/Data Out 13
//     PlcTask Outputs/GVL_iXlinker.Device_1_EtherCAT.Term_1_EK1200.Term_2_EL6002.COM_RxPDO_Map_Outputs_Channel_2.Data_Out[14] <-> COM RxPDO-Map Outputs Channel 2/Data Out 14
//     PlcTask Outputs/GVL_iXlinker.Device_1_EtherCAT.Term_1_EK1200.Term_2_EL6002.COM_RxPDO_Map_Outputs_Channel_2.Data_Out[15] <-> COM RxPDO-Map Outputs Channel 2/Data Out 15
//     PlcTask Outputs/GVL_iXlinker.Device_1_EtherCAT.Term_1_EK1200.Term_2_EL6002.COM_RxPDO_Map_Outputs_Channel_2.Data_Out[16] <-> COM RxPDO-Map Outputs Channel 2/Data Out 16
//     PlcTask Outputs/GVL_iXlinker.Device_1_EtherCAT.Term_1_EK1200.Term_2_EL6002.COM_RxPDO_Map_Outputs_Channel_2.Data_Out[17] <-> COM RxPDO-Map Outputs Channel 2/Data Out 17
//     PlcTask Outputs/GVL_iXlinker.Device_1_EtherCAT.Term_1_EK1200.Term_2_EL6002.COM_RxPDO_Map_Outputs_Channel_2.Data_Out[18] <-> COM RxPDO-Map Outputs Channel 2/Data Out 18
//     PlcTask Outputs/GVL_iXlinker.Device_1_EtherCAT.Term_1_EK1200.Term_2_EL6002.COM_RxPDO_Map_Outputs_Channel_2.Data_Out[19] <-> COM RxPDO-Map Outputs Channel 2/Data Out 19
//     PlcTask Outputs/GVL_iXlinker.Device_1_EtherCAT.Term_1_EK1200.Term_2_EL6002.COM_RxPDO_Map_Outputs_Channel_2.Data_Out[1] <-> COM RxPDO-Map Outputs Channel 2/Data Out 1
//     PlcTask Outputs/GVL_iXlinker.Device_1_EtherCAT.Term_1_EK1200.Term_2_EL6002.COM_RxPDO_Map_Outputs_Channel_2.Data_Out[20] <-> COM RxPDO-Map Outputs Channel 2/Data Out 20
//     PlcTask Outputs/GVL_iXlinker.Device_1_EtherCAT.Term_1_EK1200.Term_2_EL6002.COM_RxPDO_Map_Outputs_Channel_2.Data_Out[21] <-> COM RxPDO-Map Outputs Channel 2/Data Out 21
//     PlcTask Outputs/GVL_iXlinker.Device_1_EtherCAT.Term_1_EK1200.Term_2_EL6002.COM_RxPDO_Map_Outputs_Channel_2.Data_Out[2] <-> COM RxPDO-Map Outputs Channel 2/Data Out 2
//     PlcTask Outputs/GVL_iXlinker.Device_1_EtherCAT.Term_1_EK1200.Term_2_EL6002.COM_RxPDO_Map_Outputs_Channel_2.Data_Out[3] <-> COM RxPDO-Map Outputs Channel 2/Data Out 3
//     PlcTask Outputs/GVL_iXlinker.Device_1_EtherCAT.Term_1_EK1200.Term_2_EL6002.COM_RxPDO_Map_Outputs_Channel_2.Data_Out[4] <-> COM RxPDO-Map Outputs Channel 2/Data Out 4
//     PlcTask Outputs/GVL_iXlinker.Device_1_EtherCAT.Term_1_EK1200.Term_2_EL6002.COM_RxPDO_Map_Outputs_Channel_2.Data_Out[5] <-> COM RxPDO-Map Outputs Channel 2/Data Out 5
//     PlcTask Outputs/GVL_iXlinker.Device_1_EtherCAT.Term_1_EK1200.Term_2_EL6002.COM_RxPDO_Map_Outputs_Channel_2.Data_Out[6] <-> COM RxPDO-Map Outputs Channel 2/Data Out 6
//     PlcTask Outputs/GVL_iXlinker.Device_1_EtherCAT.Term_1_EK1200.Term_2_EL6002.COM_RxPDO_Map_Outputs_Channel_2.Data_Out[7] <-> COM RxPDO-Map Outputs Channel 2/Data Out 7
//     PlcTask Outputs/GVL_iXlinker.Device_1_EtherCAT.Term_1_EK1200.Term_2_EL6002.COM_RxPDO_Map_Outputs_Channel_2.Data_Out[8] <-> COM RxPDO-Map Outputs Channel 2/Data Out 8
//     PlcTask Outputs/GVL_iXlinker.Device_1_EtherCAT.Term_1_EK1200.Term_2_EL6002.COM_RxPDO_Map_Outputs_Channel_2.Data_Out[9] <-> COM RxPDO-Map Outputs Channel 2/Data Out 9
//   Plc1/Plc1 Instance <-> Device 1 (EtherCAT)/Term 1 (EK1200)/Term 3 (EL1809)
//     PlcTask Inputs/GVL_iXlinker.Device_1_EtherCAT.Term_1_EK1200.Term_3_EL1809.Channel_{1..16}.Input <-> Channel {1..16}/Input  (16 links)
//     PlcTask Inputs/GVL_iXlinker.Device_1_EtherCAT.Term_1_EK1200.Term_3_EL1809.InfoData.State <-> InfoData/State
//     PlcTask Inputs/GVL_iXlinker.Device_1_EtherCAT.Term_1_EK1200.Term_3_EL1809.WcState.InputToggle <-> WcState/InputToggle
//     PlcTask Inputs/GVL_iXlinker.Device_1_EtherCAT.Term_1_EK1200.Term_3_EL1809.WcState.WcState <-> WcState/WcState
//   Plc1/Plc1 Instance <-> Device 1 (EtherCAT)/Term 1 (EK1200)/Term 4 (EL2809)
//     PlcTask Inputs/GVL_iXlinker.Device_1_EtherCAT.Term_1_EK1200.Term_4_EL2809.InfoData.State <-> InfoData/State
//     PlcTask Inputs/GVL_iXlinker.Device_1_EtherCAT.Term_1_EK1200.Term_4_EL2809.WcState.WcState <-> WcState/WcState
//     PlcTask Outputs/GVL_iXlinker.Device_1_EtherCAT.Term_1_EK1200.Term_4_EL2809.Channel_{1..16}.Output <-> Channel {1..16}/Output  (16 links)
//   Plc1/Plc1 Instance <-> Device 1 (EtherCAT)/Term 1 (EK1200)/Term 5 (EL4004)
//     PlcTask Inputs/GVL_iXlinker.Device_1_EtherCAT.Term_1_EK1200.Term_5_EL4004.InfoData.AdsAddr <-> InfoData/AdsAddr
//     PlcTask Inputs/GVL_iXlinker.Device_1_EtherCAT.Term_1_EK1200.Term_5_EL4004.InfoData.State <-> InfoData/State
//     PlcTask Inputs/GVL_iXlinker.Device_1_EtherCAT.Term_1_EK1200.Term_5_EL4004.WcState.WcState <-> WcState/WcState
//     PlcTask Outputs/GVL_iXlinker.Device_1_EtherCAT.Term_1_EK1200.Term_5_EL4004.AO_Outputs_Channel_{1..4}.Analog_output <-> AO Outputs Channel {1..4}/Analog output  (4 links)
//   Plc1/Plc1 Instance <-> Device 1 (EtherCAT)/Term 1 (EK1200)/Term 6 (EL2809)
//     PlcTask Inputs/GVL_iXlinker.Device_1_EtherCAT.Term_1_EK1200.Term_6_EL2809.InfoData.State <-> InfoData/State
//     PlcTask Inputs/GVL_iXlinker.Device_1_EtherCAT.Term_1_EK1200.Term_6_EL2809.WcState.WcState <-> WcState/WcState
//     PlcTask Outputs/GVL_iXlinker.Device_1_EtherCAT.Term_1_EK1200.Term_6_EL2809.Channel_{1..16}.Output <-> Channel {1..16}/Output  (16 links)
//   Plc1/Plc1 Instance <-> Device 1 (EtherCAT)/Term 1 (EK1200)/Term 7 (EL6001)
//     PlcTask Inputs/GVL_iXlinker.Device_1_EtherCAT.Term_1_EK1200.Term_7_EL6001.COM_Inputs.Data_In[{0..21}] <-> COM Inputs/Data In {0..21}  (22 links)
//     PlcTask Inputs/GVL_iXlinker.Device_1_EtherCAT.Term_1_EK1200.Term_7_EL6001.COM_Inputs.Status/Buffer_full <-> COM Inputs/Status/Buffer full
//     PlcTask Inputs/GVL_iXlinker.Device_1_EtherCAT.Term_1_EK1200.Term_7_EL6001.COM_Inputs.Status/Framing_error <-> COM Inputs/Status/Framing error
//     PlcTask Inputs/GVL_iXlinker.Device_1_EtherCAT.Term_1_EK1200.Term_7_EL6001.COM_Inputs.Status/Init_accepted <-> COM Inputs/Status/Init accepted
//     PlcTask Inputs/GVL_iXlinker.Device_1_EtherCAT.Term_1_EK1200.Term_7_EL6001.COM_Inputs.Status/Input_length <-> COM Inputs/Status/Input length
//     PlcTask Inputs/GVL_iXlinker.Device_1_EtherCAT.Term_1_EK1200.Term_7_EL6001.COM_Inputs.Status/Overrun_error <-> COM Inputs/Status/Overrun error
//     PlcTask Inputs/GVL_iXlinker.Device_1_EtherCAT.Term_1_EK1200.Term_7_EL6001.COM_Inputs.Status/Parity_error <-> COM Inputs/Status/Parity error
//     PlcTask Inputs/GVL_iXlinker.Device_1_EtherCAT.Term_1_EK1200.Term_7_EL6001.COM_Inputs.Status/Receive_request <-> COM Inputs/Status/Receive request
//     PlcTask Inputs/GVL_iXlinker.Device_1_EtherCAT.Term_1_EK1200.Term_7_EL6001.COM_Inputs.Status/Transmit_accepted <-> COM Inputs/Status/Transmit accepted
//     PlcTask Inputs/GVL_iXlinker.Device_1_EtherCAT.Term_1_EK1200.Term_7_EL6001.InfoData.AdsAddr <-> InfoData/AdsAddr
//     PlcTask Inputs/GVL_iXlinker.Device_1_EtherCAT.Term_1_EK1200.Term_7_EL6001.InfoData.State <-> InfoData/State
//     PlcTask Inputs/GVL_iXlinker.Device_1_EtherCAT.Term_1_EK1200.Term_7_EL6001.WcState.InputToggle <-> WcState/InputToggle
//     PlcTask Inputs/GVL_iXlinker.Device_1_EtherCAT.Term_1_EK1200.Term_7_EL6001.WcState.WcState <-> WcState/WcState
//     PlcTask Outputs/GVL_iXlinker.Device_1_EtherCAT.Term_1_EK1200.Term_7_EL6001.COM_Outputs.Ctrl/Init_request <-> COM Outputs/Ctrl/Init request
//     PlcTask Outputs/GVL_iXlinker.Device_1_EtherCAT.Term_1_EK1200.Term_7_EL6001.COM_Outputs.Ctrl/Output_length <-> COM Outputs/Ctrl/Output length
//     PlcTask Outputs/GVL_iXlinker.Device_1_EtherCAT.Term_1_EK1200.Term_7_EL6001.COM_Outputs.Ctrl/Receive_accepted <-> COM Outputs/Ctrl/Receive accepted
//     PlcTask Outputs/GVL_iXlinker.Device_1_EtherCAT.Term_1_EK1200.Term_7_EL6001.COM_Outputs.Ctrl/Send_continues <-> COM Outputs/Ctrl/Send continues
//     PlcTask Outputs/GVL_iXlinker.Device_1_EtherCAT.Term_1_EK1200.Term_7_EL6001.COM_Outputs.Ctrl/Transmit_request <-> COM Outputs/Ctrl/Transmit request
//     PlcTask Outputs/GVL_iXlinker.Device_1_EtherCAT.Term_1_EK1200.Term_7_EL6001.COM_Outputs.Data_Out[{0..21}] <-> COM Outputs/Data Out {0..21}  (22 links)
//   Plc1/Plc1 Instance <-> Device 2 (EtherCAT)
//     PlcTask Inputs/GVL_iXlinker.Device_2_EtherCAT.InfoData.AmsNetId <-> InfoData/AmsNetId
//     PlcTask Inputs/GVL_iXlinker.Device_2_EtherCAT.InfoData.CfgSlaveCount <-> InfoData/CfgSlaveCount
//     PlcTask Inputs/GVL_iXlinker.Device_2_EtherCAT.InfoData.ChangeCount <-> InfoData/ChangeCount
//     PlcTask Inputs/GVL_iXlinker.Device_2_EtherCAT.InfoData.DevId <-> InfoData/DevId
//     PlcTask Inputs/GVL_iXlinker.Device_2_EtherCAT.Inputs.DevState <-> Inputs/DevState
//     PlcTask Inputs/GVL_iXlinker.Device_2_EtherCAT.Inputs.Frm0InputToggle <-> Inputs/Frm0InputToggle
//     PlcTask Inputs/GVL_iXlinker.Device_2_EtherCAT.Inputs.Frm0State <-> Inputs/Frm0State
//     PlcTask Inputs/GVL_iXlinker.Device_2_EtherCAT.Inputs.Frm0WcState <-> Inputs/Frm0WcState
//     PlcTask Inputs/GVL_iXlinker.Device_2_EtherCAT.Inputs.SlaveCount <-> Inputs/SlaveCount
//     PlcTask Inputs/GVL_iXlinker.Device_2_EtherCAT.SyncUnits.Row_{0..4}.PlcTask.InfoData.ObjectId <-> SyncUnits/Row_{0..4}/PlcTask/InfoData/ObjectId  (5 links)
//     PlcTask Inputs/GVL_iXlinker.Device_2_EtherCAT.SyncUnits.Row_{0..4}.PlcTask.InfoData.SlaveCount <-> SyncUnits/Row_{0..4}/PlcTask/InfoData/SlaveCount  (5 links)
//     PlcTask Inputs/GVL_iXlinker.Device_2_EtherCAT.SyncUnits.Row_{0..4}.PlcTask.InfoData.State <-> SyncUnits/Row_{0..4}/PlcTask/InfoData/State  (5 links)
//     PlcTask Inputs/GVL_iXlinker.Device_2_EtherCAT.SyncUnits.Row_{0..4}.PlcTask.WcState.WcState <-> SyncUnits/Row_{0..4}/PlcTask/WcState/WcState  (5 links)
//     PlcTask Inputs/GVL_iXlinker.Device_2_EtherCAT.SyncUnits._default.PlcTask.InfoData.ObjectId <-> SyncUnits/<default>/PlcTask/InfoData/ObjectId
//     PlcTask Inputs/GVL_iXlinker.Device_2_EtherCAT.SyncUnits._default.PlcTask.InfoData.SlaveCount <-> SyncUnits/<default>/PlcTask/InfoData/SlaveCount
//     PlcTask Inputs/GVL_iXlinker.Device_2_EtherCAT.SyncUnits._default.PlcTask.InfoData.State <-> SyncUnits/<default>/PlcTask/InfoData/State
//     PlcTask Inputs/GVL_iXlinker.Device_2_EtherCAT.SyncUnits._default.PlcTask.WcState.WcState <-> SyncUnits/<default>/PlcTask/WcState/WcState
//     PlcTask Outputs/GVL_iXlinker.Device_2_EtherCAT.Outputs.DevCtrl <-> Outputs/DevCtrl
//     PlcTask Outputs/GVL_iXlinker.Device_2_EtherCAT.Outputs.Frm0Ctrl <-> Outputs/Frm0Ctrl
//     PlcTask Outputs/GVL_iXlinker.Device_2_EtherCAT.Outputs.Frm0WcCtrl <-> Outputs/Frm0WcCtrl
//   Plc1/Plc1 Instance <-> Device 2 (EtherCAT)/Term 9 (EK1100)
//     PlcTask Inputs/GVL_iXlinker.Device_2_EtherCAT.Term_9_EK1100.InfoData.State <-> InfoData/State
//   Plc1/Plc1 Instance <-> Device 2 (EtherCAT)/Term 9 (EK1100)/Term 10 (EK1122)
//     PlcTask Inputs/GVL_iXlinker.Device_2_EtherCAT.Term_9_EK1100.Term_10_EK1122.InfoData.State <-> InfoData/State
//   Plc1/Plc1 Instance <-> Device 2 (EtherCAT)/Term 9 (EK1100)/Term 10 (EK1122)/Term 11 (EK1100)
//     PlcTask Inputs/GVL_iXlinker.Device_2_EtherCAT.Term_9_EK1100.Term_10_EK1122.Term_11_EK1100.InfoData.State <-> InfoData/State
//   Plc1/Plc1 Instance <-> Device 2 (EtherCAT)/Term 9 (EK1100)/Term 10 (EK1122)/Term 11 (EK1100)/Term 12 (EL3174-0002)
//     PlcTask Inputs/GVL_iXlinker.Device_2_EtherCAT.Term_9_EK1100.Term_10_EK1122.Term_11_EK1100.Term_12_EL3174_0002.AI_Standard_Channel_1.Status/Error <-> AI Standard Channel 1/Status/Error
//     PlcTask Inputs/GVL_iXlinker.Device_2_EtherCAT.Term_9_EK1100.Term_10_EK1122.Term_11_EK1100.Term_12_EL3174_0002.AI_Standard_Channel_2.Status/Error <-> AI Standard Channel 2/Status/Error
//     PlcTask Inputs/GVL_iXlinker.Device_2_EtherCAT.Term_9_EK1100.Term_10_EK1122.Term_11_EK1100.Term_12_EL3174_0002.AI_Standard_Channel_3.Status/Error <-> AI Standard Channel 3/Status/Error
//     PlcTask Inputs/GVL_iXlinker.Device_2_EtherCAT.Term_9_EK1100.Term_10_EK1122.Term_11_EK1100.Term_12_EL3174_0002.AI_Standard_Channel_4.Status/Error <-> AI Standard Channel 4/Status/Error
//     PlcTask Inputs/GVL_iXlinker.Device_2_EtherCAT.Term_9_EK1100.Term_10_EK1122.Term_11_EK1100.Term_12_EL3174_0002.AI_Standard_Channel_1.Status/Limit_1 <-> AI Standard Channel 1/Status/Limit 1
//     PlcTask Inputs/GVL_iXlinker.Device_2_EtherCAT.Term_9_EK1100.Term_10_EK1122.Term_11_EK1100.Term_12_EL3174_0002.AI_Standard_Channel_1.Status/Limit_2 <-> AI Standard Channel 1/Status/Limit 2
//     PlcTask Inputs/GVL_iXlinker.Device_2_EtherCAT.Term_9_EK1100.Term_10_EK1122.Term_11_EK1100.Term_12_EL3174_0002.AI_Standard_Channel_2.Status/Limit_1 <-> AI Standard Channel 2/Status/Limit 1
//     PlcTask Inputs/GVL_iXlinker.Device_2_EtherCAT.Term_9_EK1100.Term_10_EK1122.Term_11_EK1100.Term_12_EL3174_0002.AI_Standard_Channel_2.Status/Limit_2 <-> AI Standard Channel 2/Status/Limit 2
//     PlcTask Inputs/GVL_iXlinker.Device_2_EtherCAT.Term_9_EK1100.Term_10_EK1122.Term_11_EK1100.Term_12_EL3174_0002.AI_Standard_Channel_3.Status/Limit_1 <-> AI Standard Channel 3/Status/Limit 1
//     PlcTask Inputs/GVL_iXlinker.Device_2_EtherCAT.Term_9_EK1100.Term_10_EK1122.Term_11_EK1100.Term_12_EL3174_0002.AI_Standard_Channel_3.Status/Limit_2 <-> AI Standard Channel 3/Status/Limit 2
//     PlcTask Inputs/GVL_iXlinker.Device_2_EtherCAT.Term_9_EK1100.Term_10_EK1122.Term_11_EK1100.Term_12_EL3174_0002.AI_Standard_Channel_4.Status/Limit_1 <-> AI Standard Channel 4/Status/Limit 1
//     PlcTask Inputs/GVL_iXlinker.Device_2_EtherCAT.Term_9_EK1100.Term_10_EK1122.Term_11_EK1100.Term_12_EL3174_0002.AI_Standard_Channel_4.Status/Limit_2 <-> AI Standard Channel 4/Status/Limit 2
//     PlcTask Inputs/GVL_iXlinker.Device_2_EtherCAT.Term_9_EK1100.Term_10_EK1122.Term_11_EK1100.Term_12_EL3174_0002.AI_Standard_Channel_1.Status/Overrange <-> AI Standard Channel 1/Status/Overrange
//     PlcTask Inputs/GVL_iXlinker.Device_2_EtherCAT.Term_9_EK1100.Term_10_EK1122.Term_11_EK1100.Term_12_EL3174_0002.AI_Standard_Channel_2.Status/Overrange <-> AI Standard Channel 2/Status/Overrange
//     PlcTask Inputs/GVL_iXlinker.Device_2_EtherCAT.Term_9_EK1100.Term_10_EK1122.Term_11_EK1100.Term_12_EL3174_0002.AI_Standard_Channel_3.Status/Overrange <-> AI Standard Channel 3/Status/Overrange
//     PlcTask Inputs/GVL_iXlinker.Device_2_EtherCAT.Term_9_EK1100.Term_10_EK1122.Term_11_EK1100.Term_12_EL3174_0002.AI_Standard_Channel_4.Status/Overrange <-> AI Standard Channel 4/Status/Overrange
//     PlcTask Inputs/GVL_iXlinker.Device_2_EtherCAT.Term_9_EK1100.Term_10_EK1122.Term_11_EK1100.Term_12_EL3174_0002.AI_Standard_Channel_1.Status/Sync_error <-> AI Standard Channel 1/Status/Sync error
//     PlcTask Inputs/GVL_iXlinker.Device_2_EtherCAT.Term_9_EK1100.Term_10_EK1122.Term_11_EK1100.Term_12_EL3174_0002.AI_Standard_Channel_2.Status/Sync_error <-> AI Standard Channel 2/Status/Sync error
//     PlcTask Inputs/GVL_iXlinker.Device_2_EtherCAT.Term_9_EK1100.Term_10_EK1122.Term_11_EK1100.Term_12_EL3174_0002.AI_Standard_Channel_3.Status/Sync_error <-> AI Standard Channel 3/Status/Sync error
//     PlcTask Inputs/GVL_iXlinker.Device_2_EtherCAT.Term_9_EK1100.Term_10_EK1122.Term_11_EK1100.Term_12_EL3174_0002.AI_Standard_Channel_4.Status/Sync_error <-> AI Standard Channel 4/Status/Sync error
//     PlcTask Inputs/GVL_iXlinker.Device_2_EtherCAT.Term_9_EK1100.Term_10_EK1122.Term_11_EK1100.Term_12_EL3174_0002.AI_Standard_Channel_1.Status/TxPDO_State <-> AI Standard Channel 1/Status/TxPDO State
//     PlcTask Inputs/GVL_iXlinker.Device_2_EtherCAT.Term_9_EK1100.Term_10_EK1122.Term_11_EK1100.Term_12_EL3174_0002.AI_Standard_Channel_2.Status/TxPDO_State <-> AI Standard Channel 2/Status/TxPDO State
//     PlcTask Inputs/GVL_iXlinker.Device_2_EtherCAT.Term_9_EK1100.Term_10_EK1122.Term_11_EK1100.Term_12_EL3174_0002.AI_Standard_Channel_3.Status/TxPDO_State <-> AI Standard Channel 3/Status/TxPDO State
//     PlcTask Inputs/GVL_iXlinker.Device_2_EtherCAT.Term_9_EK1100.Term_10_EK1122.Term_11_EK1100.Term_12_EL3174_0002.AI_Standard_Channel_4.Status/TxPDO_State <-> AI Standard Channel 4/Status/TxPDO State
//     PlcTask Inputs/GVL_iXlinker.Device_2_EtherCAT.Term_9_EK1100.Term_10_EK1122.Term_11_EK1100.Term_12_EL3174_0002.AI_Standard_Channel_1.Status/TxPDO_Toggle <-> AI Standard Channel 1/Status/TxPDO Toggle
//     PlcTask Inputs/GVL_iXlinker.Device_2_EtherCAT.Term_9_EK1100.Term_10_EK1122.Term_11_EK1100.Term_12_EL3174_0002.AI_Standard_Channel_2.Status/TxPDO_Toggle <-> AI Standard Channel 2/Status/TxPDO Toggle
//     PlcTask Inputs/GVL_iXlinker.Device_2_EtherCAT.Term_9_EK1100.Term_10_EK1122.Term_11_EK1100.Term_12_EL3174_0002.AI_Standard_Channel_3.Status/TxPDO_Toggle <-> AI Standard Channel 3/Status/TxPDO Toggle
//     PlcTask Inputs/GVL_iXlinker.Device_2_EtherCAT.Term_9_EK1100.Term_10_EK1122.Term_11_EK1100.Term_12_EL3174_0002.AI_Standard_Channel_4.Status/TxPDO_Toggle <-> AI Standard Channel 4/Status/TxPDO Toggle
//     PlcTask Inputs/GVL_iXlinker.Device_2_EtherCAT.Term_9_EK1100.Term_10_EK1122.Term_11_EK1100.Term_12_EL3174_0002.AI_Standard_Channel_1.Status/Underrange <-> AI Standard Channel 1/Status/Underrange
//     PlcTask Inputs/GVL_iXlinker.Device_2_EtherCAT.Term_9_EK1100.Term_10_EK1122.Term_11_EK1100.Term_12_EL3174_0002.AI_Standard_Channel_2.Status/Underrange <-> AI Standard Channel 2/Status/Underrange
//     PlcTask Inputs/GVL_iXlinker.Device_2_EtherCAT.Term_9_EK1100.Term_10_EK1122.Term_11_EK1100.Term_12_EL3174_0002.AI_Standard_Channel_3.Status/Underrange <-> AI Standard Channel 3/Status/Underrange
//     PlcTask Inputs/GVL_iXlinker.Device_2_EtherCAT.Term_9_EK1100.Term_10_EK1122.Term_11_EK1100.Term_12_EL3174_0002.AI_Standard_Channel_4.Status/Underrange <-> AI Standard Channel 4/Status/Underrange
//     PlcTask Inputs/GVL_iXlinker.Device_2_EtherCAT.Term_9_EK1100.Term_10_EK1122.Term_11_EK1100.Term_12_EL3174_0002.AI_Standard_Channel_1.Value <-> AI Standard Channel 1/Value
//     PlcTask Inputs/GVL_iXlinker.Device_2_EtherCAT.Term_9_EK1100.Term_10_EK1122.Term_11_EK1100.Term_12_EL3174_0002.AI_Standard_Channel_2.Value <-> AI Standard Channel 2/Value
//     PlcTask Inputs/GVL_iXlinker.Device_2_EtherCAT.Term_9_EK1100.Term_10_EK1122.Term_11_EK1100.Term_12_EL3174_0002.AI_Standard_Channel_3.Value <-> AI Standard Channel 3/Value
//     PlcTask Inputs/GVL_iXlinker.Device_2_EtherCAT.Term_9_EK1100.Term_10_EK1122.Term_11_EK1100.Term_12_EL3174_0002.AI_Standard_Channel_4.Value <-> AI Standard Channel 4/Value
//     PlcTask Inputs/GVL_iXlinker.Device_2_EtherCAT.Term_9_EK1100.Term_10_EK1122.Term_11_EK1100.Term_12_EL3174_0002.InfoData.AdsAddr <-> InfoData/AdsAddr
//     PlcTask Inputs/GVL_iXlinker.Device_2_EtherCAT.Term_9_EK1100.Term_10_EK1122.Term_11_EK1100.Term_12_EL3174_0002.InfoData.State <-> InfoData/State
//     PlcTask Inputs/GVL_iXlinker.Device_2_EtherCAT.Term_9_EK1100.Term_10_EK1122.Term_11_EK1100.Term_12_EL3174_0002.WcState.InputToggle <-> WcState/InputToggle
//     PlcTask Inputs/GVL_iXlinker.Device_2_EtherCAT.Term_9_EK1100.Term_10_EK1122.Term_11_EK1100.Term_12_EL3174_0002.WcState.WcState <-> WcState/WcState
//   Plc1/Plc1 Instance <-> Device 2 (EtherCAT)/Term 9 (EK1100)/Term 10 (EK1122)/Term 11 (EK1100)/Term 13 (EL6001)
//     PlcTask Inputs/GVL_iXlinker.Device_2_EtherCAT.Term_9_EK1100.Term_10_EK1122.Term_11_EK1100.Term_13_EL6001.COM_Inputs.Data_In[{0..21}] <-> COM Inputs/Data In {0..21}  (22 links)
//     PlcTask Inputs/GVL_iXlinker.Device_2_EtherCAT.Term_9_EK1100.Term_10_EK1122.Term_11_EK1100.Term_13_EL6001.COM_Inputs.Status/Buffer_full <-> COM Inputs/Status/Buffer full
//     PlcTask Inputs/GVL_iXlinker.Device_2_EtherCAT.Term_9_EK1100.Term_10_EK1122.Term_11_EK1100.Term_13_EL6001.COM_Inputs.Status/Framing_error <-> COM Inputs/Status/Framing error
//     PlcTask Inputs/GVL_iXlinker.Device_2_EtherCAT.Term_9_EK1100.Term_10_EK1122.Term_11_EK1100.Term_13_EL6001.COM_Inputs.Status/Init_accepted <-> COM Inputs/Status/Init accepted
//     PlcTask Inputs/GVL_iXlinker.Device_2_EtherCAT.Term_9_EK1100.Term_10_EK1122.Term_11_EK1100.Term_13_EL6001.COM_Inputs.Status/Input_length <-> COM Inputs/Status/Input length
//     PlcTask Inputs/GVL_iXlinker.Device_2_EtherCAT.Term_9_EK1100.Term_10_EK1122.Term_11_EK1100.Term_13_EL6001.COM_Inputs.Status/Overrun_error <-> COM Inputs/Status/Overrun error
//     PlcTask Inputs/GVL_iXlinker.Device_2_EtherCAT.Term_9_EK1100.Term_10_EK1122.Term_11_EK1100.Term_13_EL6001.COM_Inputs.Status/Parity_error <-> COM Inputs/Status/Parity error
//     PlcTask Inputs/GVL_iXlinker.Device_2_EtherCAT.Term_9_EK1100.Term_10_EK1122.Term_11_EK1100.Term_13_EL6001.COM_Inputs.Status/Receive_request <-> COM Inputs/Status/Receive request
//     PlcTask Inputs/GVL_iXlinker.Device_2_EtherCAT.Term_9_EK1100.Term_10_EK1122.Term_11_EK1100.Term_13_EL6001.COM_Inputs.Status/Transmit_accepted <-> COM Inputs/Status/Transmit accepted
//     PlcTask Inputs/GVL_iXlinker.Device_2_EtherCAT.Term_9_EK1100.Term_10_EK1122.Term_11_EK1100.Term_13_EL6001.InfoData.AdsAddr <-> InfoData/AdsAddr
//     PlcTask Inputs/GVL_iXlinker.Device_2_EtherCAT.Term_9_EK1100.Term_10_EK1122.Term_11_EK1100.Term_13_EL6001.InfoData.State <-> InfoData/State
//     PlcTask Inputs/GVL_iXlinker.Device_2_EtherCAT.Term_9_EK1100.Term_10_EK1122.Term_11_EK1100.Term_13_EL6001.WcState.InputToggle <-> WcState/InputToggle
//     PlcTask Inputs/GVL_iXlinker.Device_2_EtherCAT.Term_9_EK1100.Term_10_EK1122.Term_11_EK1100.Term_13_EL6001.WcState.WcState <-> WcState/WcState
//     PlcTask Outputs/GVL_iXlinker.Device_2_EtherCAT.Term_9_EK1100.Term_10_EK1122.Term_11_EK1100.Term_13_EL6001.COM_Outputs.Ctrl/Init_request <-> COM Outputs/Ctrl/Init request
//     PlcTask Outputs/GVL_iXlinker.Device_2_EtherCAT.Term_9_EK1100.Term_10_EK1122.Term_11_EK1100.Term_13_EL6001.COM_Outputs.Ctrl/Output_length <-> COM Outputs/Ctrl/Output length
//     PlcTask Outputs/GVL_iXlinker.Device_2_EtherCAT.Term_9_EK1100.Term_10_EK1122.Term_11_EK1100.Term_13_EL6001.COM_Outputs.Ctrl/Receive_accepted <-> COM Outputs/Ctrl/Receive accepted
//     PlcTask Outputs/GVL_iXlinker.Device_2_EtherCAT.Term_9_EK1100.Term_10_EK1122.Term_11_EK1100.Term_13_EL6001.COM_Outputs.Ctrl/Send_continues <-> COM Outputs/Ctrl/Send continues
//     PlcTask Outputs/GVL_iXlinker.Device_2_EtherCAT.Term_9_EK1100.Term_10_EK1122.Term_11_EK1100.Term_13_EL6001.COM_Outputs.Ctrl/Transmit_request <-> COM Outputs/Ctrl/Transmit request
//     PlcTask Outputs/GVL_iXlinker.Device_2_EtherCAT.Term_9_EK1100.Term_10_EK1122.Term_11_EK1100.Term_13_EL6001.COM_Outputs.Data_Out[{0..21}] <-> COM Outputs/Data Out {0..21}  (22 links)
//   Plc1/Plc1 Instance <-> Device 2 (EtherCAT)/Term 9 (EK1100)/Term 10 (EK1122)/Term 11 (EK1100)/Term 14 (EL3011)
//     PlcTask Inputs/GVL_iXlinker.Device_2_EtherCAT.Term_9_EK1100.Term_10_EK1122.Term_11_EK1100.Term_14_EL3011.AI_Standard.Status/Error <-> AI Standard/Status/Error
//     PlcTask Inputs/GVL_iXlinker.Device_2_EtherCAT.Term_9_EK1100.Term_10_EK1122.Term_11_EK1100.Term_14_EL3011.AI_Standard.Status/Limit_1 <-> AI Standard/Status/Limit 1
//     PlcTask Inputs/GVL_iXlinker.Device_2_EtherCAT.Term_9_EK1100.Term_10_EK1122.Term_11_EK1100.Term_14_EL3011.AI_Standard.Status/Limit_2 <-> AI Standard/Status/Limit 2
//     PlcTask Inputs/GVL_iXlinker.Device_2_EtherCAT.Term_9_EK1100.Term_10_EK1122.Term_11_EK1100.Term_14_EL3011.AI_Standard.Status/Overrange <-> AI Standard/Status/Overrange
//     PlcTask Inputs/GVL_iXlinker.Device_2_EtherCAT.Term_9_EK1100.Term_10_EK1122.Term_11_EK1100.Term_14_EL3011.AI_Standard.Status/TxPDO_State <-> AI Standard/Status/TxPDO State
//     PlcTask Inputs/GVL_iXlinker.Device_2_EtherCAT.Term_9_EK1100.Term_10_EK1122.Term_11_EK1100.Term_14_EL3011.AI_Standard.Status/TxPDO_Toggle <-> AI Standard/Status/TxPDO Toggle
//     PlcTask Inputs/GVL_iXlinker.Device_2_EtherCAT.Term_9_EK1100.Term_10_EK1122.Term_11_EK1100.Term_14_EL3011.AI_Standard.Status/Underrange <-> AI Standard/Status/Underrange
//     PlcTask Inputs/GVL_iXlinker.Device_2_EtherCAT.Term_9_EK1100.Term_10_EK1122.Term_11_EK1100.Term_14_EL3011.AI_Standard.Value <-> AI Standard/Value
//     PlcTask Inputs/GVL_iXlinker.Device_2_EtherCAT.Term_9_EK1100.Term_10_EK1122.Term_11_EK1100.Term_14_EL3011.InfoData.AdsAddr <-> InfoData/AdsAddr
//     PlcTask Inputs/GVL_iXlinker.Device_2_EtherCAT.Term_9_EK1100.Term_10_EK1122.Term_11_EK1100.Term_14_EL3011.InfoData.State <-> InfoData/State
//     PlcTask Inputs/GVL_iXlinker.Device_2_EtherCAT.Term_9_EK1100.Term_10_EK1122.Term_11_EK1100.Term_14_EL3011.WcState.InputToggle <-> WcState/InputToggle
//     PlcTask Inputs/GVL_iXlinker.Device_2_EtherCAT.Term_9_EK1100.Term_10_EK1122.Term_11_EK1100.Term_14_EL3011.WcState.WcState <-> WcState/WcState
//   Plc1/Plc1 Instance <-> Device 2 (EtherCAT)/Term 9 (EK1100)/Term 10 (EK1122)/Term 11 (EK1100)/Term 15 (EL2008)
//     PlcTask Inputs/GVL_iXlinker.Device_2_EtherCAT.Term_9_EK1100.Term_10_EK1122.Term_11_EK1100.Term_15_EL2008.InfoData.State <-> InfoData/State
//     PlcTask Inputs/GVL_iXlinker.Device_2_EtherCAT.Term_9_EK1100.Term_10_EK1122.Term_11_EK1100.Term_15_EL2008.WcState.WcState <-> WcState/WcState
//     PlcTask Outputs/GVL_iXlinker.Device_2_EtherCAT.Term_9_EK1100.Term_10_EK1122.Term_11_EK1100.Term_15_EL2008.Channel_{1..8}.Output <-> Channel {1..8}/Output  (8 links)
//   Plc1/Plc1 Instance <-> Device 2 (EtherCAT)/Term 9 (EK1100)/Term 10 (EK1122)/Term 11 (EK1100)/Term 16 (EL2008)
//     PlcTask Inputs/GVL_iXlinker.Device_2_EtherCAT.Term_9_EK1100.Term_10_EK1122.Term_11_EK1100.Term_16_EL2008.InfoData.State <-> InfoData/State
//     PlcTask Inputs/GVL_iXlinker.Device_2_EtherCAT.Term_9_EK1100.Term_10_EK1122.Term_11_EK1100.Term_16_EL2008.WcState.WcState <-> WcState/WcState
//     PlcTask Outputs/GVL_iXlinker.Device_2_EtherCAT.Term_9_EK1100.Term_10_EK1122.Term_11_EK1100.Term_16_EL2008.Channel_{1..8}.Output <-> Channel {1..8}/Output  (8 links)
//   Plc1/Plc1 Instance <-> Device 2 (EtherCAT)/Term 9 (EK1100)/Term 10 (EK1122)/Term 11 (EK1100)/Term 17 (EK1110)
//     PlcTask Inputs/GVL_iXlinker.Device_2_EtherCAT.Term_9_EK1100.Term_10_EK1122.Term_11_EK1100.Term_17_EK1110.InfoData.State <-> InfoData/State
//   Plc1/Plc1 Instance <-> Device 2 (EtherCAT)/Term 9 (EK1100)/Term 10 (EK1122)/Term 18 (EK1100)
//     PlcTask Inputs/GVL_iXlinker.Device_2_EtherCAT.Term_9_EK1100.Term_10_EK1122.Term_18_EK1100.InfoData.State <-> InfoData/State
//   Plc1/Plc1 Instance <-> Device 2 (EtherCAT)/Term 9 (EK1100)/Term 10 (EK1122)/Term 18 (EK1100)/Term 19 (EL1809)
//     PlcTask Inputs/GVL_iXlinker.Device_2_EtherCAT.Term_9_EK1100.Term_10_EK1122.Term_18_EK1100.Term_19_EL1809.Channel_{1..16}.Input <-> Channel {1..16}/Input  (16 links)
//     PlcTask Inputs/GVL_iXlinker.Device_2_EtherCAT.Term_9_EK1100.Term_10_EK1122.Term_18_EK1100.Term_19_EL1809.InfoData.State <-> InfoData/State
//     PlcTask Inputs/GVL_iXlinker.Device_2_EtherCAT.Term_9_EK1100.Term_10_EK1122.Term_18_EK1100.Term_19_EL1809.WcState.InputToggle <-> WcState/InputToggle
//     PlcTask Inputs/GVL_iXlinker.Device_2_EtherCAT.Term_9_EK1100.Term_10_EK1122.Term_18_EK1100.Term_19_EL1809.WcState.WcState <-> WcState/WcState
//   Plc1/Plc1 Instance <-> Device 2 (EtherCAT)/Term 9 (EK1100)/Term 10 (EK1122)/Term 18 (EK1100)/Term 20 (EL2809)
//     PlcTask Inputs/GVL_iXlinker.Device_2_EtherCAT.Term_9_EK1100.Term_10_EK1122.Term_18_EK1100.Term_20_EL2809.InfoData.State <-> InfoData/State
//     PlcTask Inputs/GVL_iXlinker.Device_2_EtherCAT.Term_9_EK1100.Term_10_EK1122.Term_18_EK1100.Term_20_EL2809.WcState.WcState <-> WcState/WcState
//     PlcTask Outputs/GVL_iXlinker.Device_2_EtherCAT.Term_9_EK1100.Term_10_EK1122.Term_18_EK1100.Term_20_EL2809.Channel_{1..16}.Output <-> Channel {1..16}/Output  (16 links)
//   Plc1/Plc1 Instance <-> Device 2 (EtherCAT)/Term 9 (EK1100)/Term 10 (EK1122)/Term 18 (EK1100)/Term 21 (EL1809)
//     PlcTask Inputs/GVL_iXlinker.Device_2_EtherCAT.Term_9_EK1100.Term_10_EK1122.Term_18_EK1100.Term_21_EL1809.Channel_{1..16}.Input <-> Channel {1..16}/Input  (16 links)
//     PlcTask Inputs/GVL_iXlinker.Device_2_EtherCAT.Term_9_EK1100.Term_10_EK1122.Term_18_EK1100.Term_21_EL1809.InfoData.State <-> InfoData/State
//     PlcTask Inputs/GVL_iXlinker.Device_2_EtherCAT.Term_9_EK1100.Term_10_EK1122.Term_18_EK1100.Term_21_EL1809.WcState.InputToggle <-> WcState/InputToggle
//     PlcTask Inputs/GVL_iXlinker.Device_2_EtherCAT.Term_9_EK1100.Term_10_EK1122.Term_18_EK1100.Term_21_EL1809.WcState.WcState <-> WcState/WcState
//   Plc1/Plc1 Instance <-> Device 2 (EtherCAT)/Term 9 (EK1100)/Term 10 (EK1122)/Term 18 (EK1100)/Term 22 (EL3011)
//     PlcTask Inputs/GVL_iXlinker.Device_2_EtherCAT.Term_9_EK1100.Term_10_EK1122.Term_18_EK1100.Term_22_EL3011.AI_Standard.Status/Error <-> AI Standard/Status/Error
//     PlcTask Inputs/GVL_iXlinker.Device_2_EtherCAT.Term_9_EK1100.Term_10_EK1122.Term_18_EK1100.Term_22_EL3011.AI_Standard.Status/Limit_1 <-> AI Standard/Status/Limit 1
//     PlcTask Inputs/GVL_iXlinker.Device_2_EtherCAT.Term_9_EK1100.Term_10_EK1122.Term_18_EK1100.Term_22_EL3011.AI_Standard.Status/Limit_2 <-> AI Standard/Status/Limit 2
//     PlcTask Inputs/GVL_iXlinker.Device_2_EtherCAT.Term_9_EK1100.Term_10_EK1122.Term_18_EK1100.Term_22_EL3011.AI_Standard.Status/Overrange <-> AI Standard/Status/Overrange
//     PlcTask Inputs/GVL_iXlinker.Device_2_EtherCAT.Term_9_EK1100.Term_10_EK1122.Term_18_EK1100.Term_22_EL3011.AI_Standard.Status/TxPDO_State <-> AI Standard/Status/TxPDO State
//     PlcTask Inputs/GVL_iXlinker.Device_2_EtherCAT.Term_9_EK1100.Term_10_EK1122.Term_18_EK1100.Term_22_EL3011.AI_Standard.Status/TxPDO_Toggle <-> AI Standard/Status/TxPDO Toggle
//     PlcTask Inputs/GVL_iXlinker.Device_2_EtherCAT.Term_9_EK1100.Term_10_EK1122.Term_18_EK1100.Term_22_EL3011.AI_Standard.Status/Underrange <-> AI Standard/Status/Underrange
//     PlcTask Inputs/GVL_iXlinker.Device_2_EtherCAT.Term_9_EK1100.Term_10_EK1122.Term_18_EK1100.Term_22_EL3011.AI_Standard.Value <-> AI Standard/Value
//     PlcTask Inputs/GVL_iXlinker.Device_2_EtherCAT.Term_9_EK1100.Term_10_EK1122.Term_18_EK1100.Term_22_EL3011.InfoData.AdsAddr <-> InfoData/AdsAddr
//     PlcTask Inputs/GVL_iXlinker.Device_2_EtherCAT.Term_9_EK1100.Term_10_EK1122.Term_18_EK1100.Term_22_EL3011.InfoData.State <-> InfoData/State
//     PlcTask Inputs/GVL_iXlinker.Device_2_EtherCAT.Term_9_EK1100.Term_10_EK1122.Term_18_EK1100.Term_22_EL3011.WcState.InputToggle <-> WcState/InputToggle
//     PlcTask Inputs/GVL_iXlinker.Device_2_EtherCAT.Term_9_EK1100.Term_10_EK1122.Term_18_EK1100.Term_22_EL3011.WcState.WcState <-> WcState/WcState
//   Plc1/Plc1 Instance <-> Device 2 (EtherCAT)/Term 9 (EK1100)/Term 10 (EK1122)/Term 23 (EK1100)
//     PlcTask Inputs/GVL_iXlinker.Device_2_EtherCAT.Term_9_EK1100.Term_10_EK1122.Term_23_EK1100.InfoData.State <-> InfoData/State
//   Plc1/Plc1 Instance <-> Device 2 (EtherCAT)/Term 9 (EK1100)/Term 10 (EK1122)/Term 23 (EK1100)/Term 24 (EK1122)
//     PlcTask Inputs/GVL_iXlinker.Device_2_EtherCAT.Term_9_EK1100.Term_10_EK1122.Term_23_EK1100.Term_24_EK1122.InfoData.State <-> InfoData/State
//   Plc1/Plc1 Instance <-> Device 2 (EtherCAT)/Term 9 (EK1100)/Term 10 (EK1122)/Term 23 (EK1100)/Term 24 (EK1122)/Term 25 (EK1100)
//     PlcTask Inputs/GVL_iXlinker.Device_2_EtherCAT.Term_9_EK1100.Term_10_EK1122.Term_23_EK1100.Term_24_EK1122.Term_25_EK1100.InfoData.State <-> InfoData/State
//   Plc1/Plc1 Instance <-> Device 2 (EtherCAT)/Term 9 (EK1100)/Term 10 (EK1122)/Term 23 (EK1100)/Term 24 (EK1122)/Term 25 (EK1100)/Term 26 (EL1819)
//     PlcTask Inputs/GVL_iXlinker.Device_2_EtherCAT.Term_9_EK1100.Term_10_EK1122.Term_23_EK1100.Term_24_EK1122.Term_25_EK1100.Term_26_EL1819.Channel_{1..16}.Input <-> Channel {1..16}/Input  (16 links)
//     PlcTask Inputs/GVL_iXlinker.Device_2_EtherCAT.Term_9_EK1100.Term_10_EK1122.Term_23_EK1100.Term_24_EK1122.Term_25_EK1100.Term_26_EL1819.InfoData.State <-> InfoData/State
//     PlcTask Inputs/GVL_iXlinker.Device_2_EtherCAT.Term_9_EK1100.Term_10_EK1122.Term_23_EK1100.Term_24_EK1122.Term_25_EK1100.Term_26_EL1819.WcState.InputToggle <-> WcState/InputToggle
//     PlcTask Inputs/GVL_iXlinker.Device_2_EtherCAT.Term_9_EK1100.Term_10_EK1122.Term_23_EK1100.Term_24_EK1122.Term_25_EK1100.Term_26_EL1819.WcState.WcState <-> WcState/WcState
//   Plc1/Plc1 Instance <-> Device 2 (EtherCAT)/Term 9 (EK1100)/Term 10 (EK1122)/Term 23 (EK1100)/Term 24 (EK1122)/Term 25 (EK1100)/Term 27 (EL1819)
//     PlcTask Inputs/GVL_iXlinker.Device_2_EtherCAT.Term_9_EK1100.Term_10_EK1122.Term_23_EK1100.Term_24_EK1122.Term_25_EK1100.Term_27_EL1819.Channel_{1..16}.Input <-> Channel {1..16}/Input  (16 links)
//     PlcTask Inputs/GVL_iXlinker.Device_2_EtherCAT.Term_9_EK1100.Term_10_EK1122.Term_23_EK1100.Term_24_EK1122.Term_25_EK1100.Term_27_EL1819.InfoData.State <-> InfoData/State
//     PlcTask Inputs/GVL_iXlinker.Device_2_EtherCAT.Term_9_EK1100.Term_10_EK1122.Term_23_EK1100.Term_24_EK1122.Term_25_EK1100.Term_27_EL1819.WcState.InputToggle <-> WcState/InputToggle
//     PlcTask Inputs/GVL_iXlinker.Device_2_EtherCAT.Term_9_EK1100.Term_10_EK1122.Term_23_EK1100.Term_24_EK1122.Term_25_EK1100.Term_27_EL1819.WcState.WcState <-> WcState/WcState
//   Plc1/Plc1 Instance <-> Device 2 (EtherCAT)/Term 9 (EK1100)/Term 10 (EK1122)/Term 23 (EK1100)/Term 24 (EK1122)/Term 28 (EK1100)
//     PlcTask Inputs/GVL_iXlinker.Device_2_EtherCAT.Term_9_EK1100.Term_10_EK1122.Term_23_EK1100.Term_24_EK1122.Term_28_EK1100.InfoData.State <-> InfoData/State
//   Plc1/Plc1 Instance <-> Device 2 (EtherCAT)/Term 9 (EK1100)/Term 10 (EK1122)/Term 23 (EK1100)/Term 24 (EK1122)/Term 28 (EK1100)/Term 29 (EL2788)
//     PlcTask Inputs/GVL_iXlinker.Device_2_EtherCAT.Term_9_EK1100.Term_10_EK1122.Term_23_EK1100.Term_24_EK1122.Term_28_EK1100.Term_29_EL2788.InfoData.State <-> InfoData/State
//     PlcTask Inputs/GVL_iXlinker.Device_2_EtherCAT.Term_9_EK1100.Term_10_EK1122.Term_23_EK1100.Term_24_EK1122.Term_28_EK1100.Term_29_EL2788.WcState.WcState <-> WcState/WcState
//     PlcTask Outputs/GVL_iXlinker.Device_2_EtherCAT.Term_9_EK1100.Term_10_EK1122.Term_23_EK1100.Term_24_EK1122.Term_28_EK1100.Term_29_EL2788.Channel_{1..8}.Output <-> Channel {1..8}/Output  (8 links)
//   Plc1/Plc1 Instance <-> Device 2 (EtherCAT)/Term 9 (EK1100)/Term 10 (EK1122)/Term 23 (EK1100)/Term 24 (EK1122)/Term 28 (EK1100)/Term 30 (EL3773)
//     PlcTask Inputs/GVL_iXlinker.Device_2_EtherCAT.Term_9_EK1100.Term_10_EK1122.Term_23_EK1100.Term_24_EK1122.Term_28_EK1100.Term_30_EL3773.AI_NextSync1Time.StartTimeNextLatch/Hi <-> AI NextSync1Time/StartTimeNextLatch/Hi
//     PlcTask Inputs/GVL_iXlinker.Device_2_EtherCAT.Term_9_EK1100.Term_10_EK1122.Term_23_EK1100.Term_24_EK1122.Term_28_EK1100.Term_30_EL3773.AI_NextSync1Time.StartTimeNextLatch/Low <-> AI NextSync1Time/StartTimeNextLatch/Low
//     PlcTask Inputs/GVL_iXlinker.Device_2_EtherCAT.Term_9_EK1100.Term_10_EK1122.Term_23_EK1100.Term_24_EK1122.Term_28_EK1100.Term_30_EL3773.AI_Sample_Count.Sample_Count <-> AI Sample Count/Sample Count
//     PlcTask Inputs/GVL_iXlinker.Device_2_EtherCAT.Term_9_EK1100.Term_10_EK1122.Term_23_EK1100.Term_24_EK1122.Term_28_EK1100.Term_30_EL3773.InfoData.AdsAddr <-> InfoData/AdsAddr
//     PlcTask Inputs/GVL_iXlinker.Device_2_EtherCAT.Term_9_EK1100.Term_10_EK1122.Term_23_EK1100.Term_24_EK1122.Term_28_EK1100.Term_30_EL3773.InfoData.DcInputShift <-> InfoData/DcInputShift
//     PlcTask Inputs/GVL_iXlinker.Device_2_EtherCAT.Term_9_EK1100.Term_10_EK1122.Term_23_EK1100.Term_24_EK1122.Term_28_EK1100.Term_30_EL3773.InfoData.DcOutputShift <-> InfoData/DcOutputShift
//     PlcTask Inputs/GVL_iXlinker.Device_2_EtherCAT.Term_9_EK1100.Term_10_EK1122.Term_23_EK1100.Term_24_EK1122.Term_28_EK1100.Term_30_EL3773.InfoData.State <-> InfoData/State
//     PlcTask Inputs/GVL_iXlinker.Device_2_EtherCAT.Term_9_EK1100.Term_10_EK1122.Term_23_EK1100.Term_24_EK1122.Term_28_EK1100.Term_30_EL3773.L1_Current_Status.I1_Status/Error <-> L1 Current Status/I1 Status/Error
//     PlcTask Inputs/GVL_iXlinker.Device_2_EtherCAT.Term_9_EK1100.Term_10_EK1122.Term_23_EK1100.Term_24_EK1122.Term_28_EK1100.Term_30_EL3773.L2_Current_Status.I2_Status/Error <-> L2 Current Status/I2 Status/Error
//     PlcTask Inputs/GVL_iXlinker.Device_2_EtherCAT.Term_9_EK1100.Term_10_EK1122.Term_23_EK1100.Term_24_EK1122.Term_28_EK1100.Term_30_EL3773.L3_Current_Status.I3_Status/Error <-> L3 Current Status/I3 Status/Error
//     PlcTask Inputs/GVL_iXlinker.Device_2_EtherCAT.Term_9_EK1100.Term_10_EK1122.Term_23_EK1100.Term_24_EK1122.Term_28_EK1100.Term_30_EL3773.L1_Current_Status.I1_Status/Limit_x <-> L1 Current Status/I1 Status/Limit
//     PlcTask Inputs/GVL_iXlinker.Device_2_EtherCAT.Term_9_EK1100.Term_10_EK1122.Term_23_EK1100.Term_24_EK1122.Term_28_EK1100.Term_30_EL3773.L2_Current_Status.I2_Status/Limit_x <-> L2 Current Status/I2 Status/Limit
//     PlcTask Inputs/GVL_iXlinker.Device_2_EtherCAT.Term_9_EK1100.Term_10_EK1122.Term_23_EK1100.Term_24_EK1122.Term_28_EK1100.Term_30_EL3773.L3_Current_Status.I3_Status/Limit_x <-> L3 Current Status/I3 Status/Limit
//     PlcTask Inputs/GVL_iXlinker.Device_2_EtherCAT.Term_9_EK1100.Term_10_EK1122.Term_23_EK1100.Term_24_EK1122.Term_28_EK1100.Term_30_EL3773.L1_Current_Status.I1_Status/Overrange <-> L1 Current Status/I1 Status/Overrange
//     PlcTask Inputs/GVL_iXlinker.Device_2_EtherCAT.Term_9_EK1100.Term_10_EK1122.Term_23_EK1100.Term_24_EK1122.Term_28_EK1100.Term_30_EL3773.L2_Current_Status.I2_Status/Overrange <-> L2 Current Status/I2 Status/Overrange
//     PlcTask Inputs/GVL_iXlinker.Device_2_EtherCAT.Term_9_EK1100.Term_10_EK1122.Term_23_EK1100.Term_24_EK1122.Term_28_EK1100.Term_30_EL3773.L3_Current_Status.I3_Status/Overrange <-> L3 Current Status/I3 Status/Overrange
//     PlcTask Inputs/GVL_iXlinker.Device_2_EtherCAT.Term_9_EK1100.Term_10_EK1122.Term_23_EK1100.Term_24_EK1122.Term_28_EK1100.Term_30_EL3773.L1_Current_Status.I1_Status/Sync_error <-> L1 Current Status/I1 Status/Sync error
//     PlcTask Inputs/GVL_iXlinker.Device_2_EtherCAT.Term_9_EK1100.Term_10_EK1122.Term_23_EK1100.Term_24_EK1122.Term_28_EK1100.Term_30_EL3773.L2_Current_Status.I2_Status/Sync_error <-> L2 Current Status/I2 Status/Sync error
//     PlcTask Inputs/GVL_iXlinker.Device_2_EtherCAT.Term_9_EK1100.Term_10_EK1122.Term_23_EK1100.Term_24_EK1122.Term_28_EK1100.Term_30_EL3773.L3_Current_Status.I3_Status/Sync_error <-> L3 Current Status/I3 Status/Sync error
//     PlcTask Inputs/GVL_iXlinker.Device_2_EtherCAT.Term_9_EK1100.Term_10_EK1122.Term_23_EK1100.Term_24_EK1122.Term_28_EK1100.Term_30_EL3773.L1_Current_Status.I1_Status/TxPDO_State <-> L1 Current Status/I1 Status/TxPDO State
//     PlcTask Inputs/GVL_iXlinker.Device_2_EtherCAT.Term_9_EK1100.Term_10_EK1122.Term_23_EK1100.Term_24_EK1122.Term_28_EK1100.Term_30_EL3773.L2_Current_Status.I2_Status/TxPDO_State <-> L2 Current Status/I2 Status/TxPDO State
//     PlcTask Inputs/GVL_iXlinker.Device_2_EtherCAT.Term_9_EK1100.Term_10_EK1122.Term_23_EK1100.Term_24_EK1122.Term_28_EK1100.Term_30_EL3773.L3_Current_Status.I3_Status/TxPDO_State <-> L3 Current Status/I3 Status/TxPDO State
//     PlcTask Inputs/GVL_iXlinker.Device_2_EtherCAT.Term_9_EK1100.Term_10_EK1122.Term_23_EK1100.Term_24_EK1122.Term_28_EK1100.Term_30_EL3773.L1_Current_Status.I1_Status/TxPDO_Toggle <-> L1 Current Status/I1 Status/TxPDO Toggle
//     PlcTask Inputs/GVL_iXlinker.Device_2_EtherCAT.Term_9_EK1100.Term_10_EK1122.Term_23_EK1100.Term_24_EK1122.Term_28_EK1100.Term_30_EL3773.L2_Current_Status.I2_Status/TxPDO_Toggle <-> L2 Current Status/I2 Status/TxPDO Toggle
//     PlcTask Inputs/GVL_iXlinker.Device_2_EtherCAT.Term_9_EK1100.Term_10_EK1122.Term_23_EK1100.Term_24_EK1122.Term_28_EK1100.Term_30_EL3773.L3_Current_Status.I3_Status/TxPDO_Toggle <-> L3 Current Status/I3 Status/TxPDO Toggle
//     PlcTask Inputs/GVL_iXlinker.Device_2_EtherCAT.Term_9_EK1100.Term_10_EK1122.Term_23_EK1100.Term_24_EK1122.Term_28_EK1100.Term_30_EL3773.L1_Current_Status.I1_Status/Underrange <-> L1 Current Status/I1 Status/Underrange
//     PlcTask Inputs/GVL_iXlinker.Device_2_EtherCAT.Term_9_EK1100.Term_10_EK1122.Term_23_EK1100.Term_24_EK1122.Term_28_EK1100.Term_30_EL3773.L2_Current_Status.I2_Status/Underrange <-> L2 Current Status/I2 Status/Underrange
//     PlcTask Inputs/GVL_iXlinker.Device_2_EtherCAT.Term_9_EK1100.Term_10_EK1122.Term_23_EK1100.Term_24_EK1122.Term_28_EK1100.Term_30_EL3773.L3_Current_Status.I3_Status/Underrange <-> L3 Current Status/I3 Status/Underrange
//     PlcTask Inputs/GVL_iXlinker.Device_2_EtherCAT.Term_9_EK1100.Term_10_EK1122.Term_23_EK1100.Term_24_EK1122.Term_28_EK1100.Term_30_EL3773.L1_Voltage_Status.U1_Status/Error <-> L1 Voltage Status/U1 Status/Error
//     PlcTask Inputs/GVL_iXlinker.Device_2_EtherCAT.Term_9_EK1100.Term_10_EK1122.Term_23_EK1100.Term_24_EK1122.Term_28_EK1100.Term_30_EL3773.L2_Voltage_Status.U2_Status/Error <-> L2 Voltage Status/U2 Status/Error
//     PlcTask Inputs/GVL_iXlinker.Device_2_EtherCAT.Term_9_EK1100.Term_10_EK1122.Term_23_EK1100.Term_24_EK1122.Term_28_EK1100.Term_30_EL3773.L3_Voltage_Status.U3_Status/Error <-> L3 Voltage Status/U3 Status/Error
//     PlcTask Inputs/GVL_iXlinker.Device_2_EtherCAT.Term_9_EK1100.Term_10_EK1122.Term_23_EK1100.Term_24_EK1122.Term_28_EK1100.Term_30_EL3773.L1_Voltage_Status.U1_Status/Limit_x <-> L1 Voltage Status/U1 Status/Limit
//     PlcTask Inputs/GVL_iXlinker.Device_2_EtherCAT.Term_9_EK1100.Term_10_EK1122.Term_23_EK1100.Term_24_EK1122.Term_28_EK1100.Term_30_EL3773.L2_Voltage_Status.U2_Status/Limit_x <-> L2 Voltage Status/U2 Status/Limit
//     PlcTask Inputs/GVL_iXlinker.Device_2_EtherCAT.Term_9_EK1100.Term_10_EK1122.Term_23_EK1100.Term_24_EK1122.Term_28_EK1100.Term_30_EL3773.L3_Voltage_Status.U3_Status/Limit_x <-> L3 Voltage Status/U3 Status/Limit
//     PlcTask Inputs/GVL_iXlinker.Device_2_EtherCAT.Term_9_EK1100.Term_10_EK1122.Term_23_EK1100.Term_24_EK1122.Term_28_EK1100.Term_30_EL3773.L1_Voltage_Status.U1_Status/Overrange <-> L1 Voltage Status/U1 Status/Overrange
//     PlcTask Inputs/GVL_iXlinker.Device_2_EtherCAT.Term_9_EK1100.Term_10_EK1122.Term_23_EK1100.Term_24_EK1122.Term_28_EK1100.Term_30_EL3773.L2_Voltage_Status.U2_Status/Overrange <-> L2 Voltage Status/U2 Status/Overrange
//     PlcTask Inputs/GVL_iXlinker.Device_2_EtherCAT.Term_9_EK1100.Term_10_EK1122.Term_23_EK1100.Term_24_EK1122.Term_28_EK1100.Term_30_EL3773.L3_Voltage_Status.U3_Status/Overrange <-> L3 Voltage Status/U3 Status/Overrange
//     PlcTask Inputs/GVL_iXlinker.Device_2_EtherCAT.Term_9_EK1100.Term_10_EK1122.Term_23_EK1100.Term_24_EK1122.Term_28_EK1100.Term_30_EL3773.L1_Voltage_Status.U1_Status/Sync_error <-> L1 Voltage Status/U1 Status/Sync error
//     PlcTask Inputs/GVL_iXlinker.Device_2_EtherCAT.Term_9_EK1100.Term_10_EK1122.Term_23_EK1100.Term_24_EK1122.Term_28_EK1100.Term_30_EL3773.L2_Voltage_Status.U2_Status/Sync_error <-> L2 Voltage Status/U2 Status/Sync error
//     PlcTask Inputs/GVL_iXlinker.Device_2_EtherCAT.Term_9_EK1100.Term_10_EK1122.Term_23_EK1100.Term_24_EK1122.Term_28_EK1100.Term_30_EL3773.L3_Voltage_Status.U3_Status/Sync_error <-> L3 Voltage Status/U3 Status/Sync error
//     PlcTask Inputs/GVL_iXlinker.Device_2_EtherCAT.Term_9_EK1100.Term_10_EK1122.Term_23_EK1100.Term_24_EK1122.Term_28_EK1100.Term_30_EL3773.L1_Voltage_Status.U1_Status/TxPDO_State <-> L1 Voltage Status/U1 Status/TxPDO State
//     PlcTask Inputs/GVL_iXlinker.Device_2_EtherCAT.Term_9_EK1100.Term_10_EK1122.Term_23_EK1100.Term_24_EK1122.Term_28_EK1100.Term_30_EL3773.L2_Voltage_Status.U2_Status/TxPDO_State <-> L2 Voltage Status/U2 Status/TxPDO State
//     PlcTask Inputs/GVL_iXlinker.Device_2_EtherCAT.Term_9_EK1100.Term_10_EK1122.Term_23_EK1100.Term_24_EK1122.Term_28_EK1100.Term_30_EL3773.L3_Voltage_Status.U3_Status/TxPDO_State <-> L3 Voltage Status/U3 Status/TxPDO State
//     PlcTask Inputs/GVL_iXlinker.Device_2_EtherCAT.Term_9_EK1100.Term_10_EK1122.Term_23_EK1100.Term_24_EK1122.Term_28_EK1100.Term_30_EL3773.L1_Voltage_Status.U1_Status/TxPDO_Toggle <-> L1 Voltage Status/U1 Status/TxPDO Toggle
//     PlcTask Inputs/GVL_iXlinker.Device_2_EtherCAT.Term_9_EK1100.Term_10_EK1122.Term_23_EK1100.Term_24_EK1122.Term_28_EK1100.Term_30_EL3773.L2_Voltage_Status.U2_Status/TxPDO_Toggle <-> L2 Voltage Status/U2 Status/TxPDO Toggle
//     PlcTask Inputs/GVL_iXlinker.Device_2_EtherCAT.Term_9_EK1100.Term_10_EK1122.Term_23_EK1100.Term_24_EK1122.Term_28_EK1100.Term_30_EL3773.L3_Voltage_Status.U3_Status/TxPDO_Toggle <-> L3 Voltage Status/U3 Status/TxPDO Toggle
//     PlcTask Inputs/GVL_iXlinker.Device_2_EtherCAT.Term_9_EK1100.Term_10_EK1122.Term_23_EK1100.Term_24_EK1122.Term_28_EK1100.Term_30_EL3773.L1_Voltage_Status.U1_Status/Underrange <-> L1 Voltage Status/U1 Status/Underrange
//     PlcTask Inputs/GVL_iXlinker.Device_2_EtherCAT.Term_9_EK1100.Term_10_EK1122.Term_23_EK1100.Term_24_EK1122.Term_28_EK1100.Term_30_EL3773.L2_Voltage_Status.U2_Status/Underrange <-> L2 Voltage Status/U2 Status/Underrange
//     PlcTask Inputs/GVL_iXlinker.Device_2_EtherCAT.Term_9_EK1100.Term_10_EK1122.Term_23_EK1100.Term_24_EK1122.Term_28_EK1100.Term_30_EL3773.L3_Voltage_Status.U3_Status/Underrange <-> L3 Voltage Status/U3 Status/Underrange
//     PlcTask Inputs/GVL_iXlinker.Device_2_EtherCAT.Term_9_EK1100.Term_10_EK1122.Term_23_EK1100.Term_24_EK1122.Term_28_EK1100.Term_30_EL3773.WcState.InputToggle <-> WcState/InputToggle
//     PlcTask Inputs/GVL_iXlinker.Device_2_EtherCAT.Term_9_EK1100.Term_10_EK1122.Term_23_EK1100.Term_24_EK1122.Term_28_EK1100.Term_30_EL3773.WcState.WcState <-> WcState/WcState
//   Plc1/Plc1 Instance <-> Device 2 (EtherCAT)/Term 9 (EK1100)/Term 10 (EK1122)/Term 23 (EK1100)/Term 31 (EL3773)
//     PlcTask Inputs/GVL_iXlinker.Device_2_EtherCAT.Term_9_EK1100.Term_10_EK1122.Term_23_EK1100.Term_31_EL3773.AI_NextSync1Time.StartTimeNextLatch/Hi <-> AI NextSync1Time/StartTimeNextLatch/Hi
//     PlcTask Inputs/GVL_iXlinker.Device_2_EtherCAT.Term_9_EK1100.Term_10_EK1122.Term_23_EK1100.Term_31_EL3773.AI_NextSync1Time.StartTimeNextLatch/Low <-> AI NextSync1Time/StartTimeNextLatch/Low
//     PlcTask Inputs/GVL_iXlinker.Device_2_EtherCAT.Term_9_EK1100.Term_10_EK1122.Term_23_EK1100.Term_31_EL3773.AI_Sample_Count.Sample_Count <-> AI Sample Count/Sample Count
//     PlcTask Inputs/GVL_iXlinker.Device_2_EtherCAT.Term_9_EK1100.Term_10_EK1122.Term_23_EK1100.Term_31_EL3773.InfoData.AdsAddr <-> InfoData/AdsAddr
//     PlcTask Inputs/GVL_iXlinker.Device_2_EtherCAT.Term_9_EK1100.Term_10_EK1122.Term_23_EK1100.Term_31_EL3773.InfoData.DcInputShift <-> InfoData/DcInputShift
//     PlcTask Inputs/GVL_iXlinker.Device_2_EtherCAT.Term_9_EK1100.Term_10_EK1122.Term_23_EK1100.Term_31_EL3773.InfoData.DcOutputShift <-> InfoData/DcOutputShift
//     PlcTask Inputs/GVL_iXlinker.Device_2_EtherCAT.Term_9_EK1100.Term_10_EK1122.Term_23_EK1100.Term_31_EL3773.InfoData.State <-> InfoData/State
//     PlcTask Inputs/GVL_iXlinker.Device_2_EtherCAT.Term_9_EK1100.Term_10_EK1122.Term_23_EK1100.Term_31_EL3773.L1_Current_Status.I1_Status/Error <-> L1 Current Status/I1 Status/Error
//     PlcTask Inputs/GVL_iXlinker.Device_2_EtherCAT.Term_9_EK1100.Term_10_EK1122.Term_23_EK1100.Term_31_EL3773.L2_Current_Status.I2_Status/Error <-> L2 Current Status/I2 Status/Error
//     PlcTask Inputs/GVL_iXlinker.Device_2_EtherCAT.Term_9_EK1100.Term_10_EK1122.Term_23_EK1100.Term_31_EL3773.L3_Current_Status.I3_Status/Error <-> L3 Current Status/I3 Status/Error
//     PlcTask Inputs/GVL_iXlinker.Device_2_EtherCAT.Term_9_EK1100.Term_10_EK1122.Term_23_EK1100.Term_31_EL3773.L1_Current_Status.I1_Status/Limit_x <-> L1 Current Status/I1 Status/Limit
//     PlcTask Inputs/GVL_iXlinker.Device_2_EtherCAT.Term_9_EK1100.Term_10_EK1122.Term_23_EK1100.Term_31_EL3773.L2_Current_Status.I2_Status/Limit_x <-> L2 Current Status/I2 Status/Limit
//     PlcTask Inputs/GVL_iXlinker.Device_2_EtherCAT.Term_9_EK1100.Term_10_EK1122.Term_23_EK1100.Term_31_EL3773.L3_Current_Status.I3_Status/Limit_x <-> L3 Current Status/I3 Status/Limit
//     PlcTask Inputs/GVL_iXlinker.Device_2_EtherCAT.Term_9_EK1100.Term_10_EK1122.Term_23_EK1100.Term_31_EL3773.L1_Current_Status.I1_Status/Overrange <-> L1 Current Status/I1 Status/Overrange
//     PlcTask Inputs/GVL_iXlinker.Device_2_EtherCAT.Term_9_EK1100.Term_10_EK1122.Term_23_EK1100.Term_31_EL3773.L2_Current_Status.I2_Status/Overrange <-> L2 Current Status/I2 Status/Overrange
//     PlcTask Inputs/GVL_iXlinker.Device_2_EtherCAT.Term_9_EK1100.Term_10_EK1122.Term_23_EK1100.Term_31_EL3773.L3_Current_Status.I3_Status/Overrange <-> L3 Current Status/I3 Status/Overrange
//     PlcTask Inputs/GVL_iXlinker.Device_2_EtherCAT.Term_9_EK1100.Term_10_EK1122.Term_23_EK1100.Term_31_EL3773.L1_Current_Status.I1_Status/Sync_error <-> L1 Current Status/I1 Status/Sync error
//     PlcTask Inputs/GVL_iXlinker.Device_2_EtherCAT.Term_9_EK1100.Term_10_EK1122.Term_23_EK1100.Term_31_EL3773.L2_Current_Status.I2_Status/Sync_error <-> L2 Current Status/I2 Status/Sync error
//     PlcTask Inputs/GVL_iXlinker.Device_2_EtherCAT.Term_9_EK1100.Term_10_EK1122.Term_23_EK1100.Term_31_EL3773.L3_Current_Status.I3_Status/Sync_error <-> L3 Current Status/I3 Status/Sync error
//     PlcTask Inputs/GVL_iXlinker.Device_2_EtherCAT.Term_9_EK1100.Term_10_EK1122.Term_23_EK1100.Term_31_EL3773.L1_Current_Status.I1_Status/TxPDO_State <-> L1 Current Status/I1 Status/TxPDO State
//     PlcTask Inputs/GVL_iXlinker.Device_2_EtherCAT.Term_9_EK1100.Term_10_EK1122.Term_23_EK1100.Term_31_EL3773.L2_Current_Status.I2_Status/TxPDO_State <-> L2 Current Status/I2 Status/TxPDO State
//     PlcTask Inputs/GVL_iXlinker.Device_2_EtherCAT.Term_9_EK1100.Term_10_EK1122.Term_23_EK1100.Term_31_EL3773.L3_Current_Status.I3_Status/TxPDO_State <-> L3 Current Status/I3 Status/TxPDO State
//     PlcTask Inputs/GVL_iXlinker.Device_2_EtherCAT.Term_9_EK1100.Term_10_EK1122.Term_23_EK1100.Term_31_EL3773.L1_Current_Status.I1_Status/TxPDO_Toggle <-> L1 Current Status/I1 Status/TxPDO Toggle
//     PlcTask Inputs/GVL_iXlinker.Device_2_EtherCAT.Term_9_EK1100.Term_10_EK1122.Term_23_EK1100.Term_31_EL3773.L2_Current_Status.I2_Status/TxPDO_Toggle <-> L2 Current Status/I2 Status/TxPDO Toggle
//     PlcTask Inputs/GVL_iXlinker.Device_2_EtherCAT.Term_9_EK1100.Term_10_EK1122.Term_23_EK1100.Term_31_EL3773.L3_Current_Status.I3_Status/TxPDO_Toggle <-> L3 Current Status/I3 Status/TxPDO Toggle
//     PlcTask Inputs/GVL_iXlinker.Device_2_EtherCAT.Term_9_EK1100.Term_10_EK1122.Term_23_EK1100.Term_31_EL3773.L1_Current_Status.I1_Status/Underrange <-> L1 Current Status/I1 Status/Underrange
//     PlcTask Inputs/GVL_iXlinker.Device_2_EtherCAT.Term_9_EK1100.Term_10_EK1122.Term_23_EK1100.Term_31_EL3773.L2_Current_Status.I2_Status/Underrange <-> L2 Current Status/I2 Status/Underrange
//     PlcTask Inputs/GVL_iXlinker.Device_2_EtherCAT.Term_9_EK1100.Term_10_EK1122.Term_23_EK1100.Term_31_EL3773.L3_Current_Status.I3_Status/Underrange <-> L3 Current Status/I3 Status/Underrange
//     PlcTask Inputs/GVL_iXlinker.Device_2_EtherCAT.Term_9_EK1100.Term_10_EK1122.Term_23_EK1100.Term_31_EL3773.L1_Voltage_Status.U1_Status/Error <-> L1 Voltage Status/U1 Status/Error
//     PlcTask Inputs/GVL_iXlinker.Device_2_EtherCAT.Term_9_EK1100.Term_10_EK1122.Term_23_EK1100.Term_31_EL3773.L2_Voltage_Status.U2_Status/Error <-> L2 Voltage Status/U2 Status/Error
//     PlcTask Inputs/GVL_iXlinker.Device_2_EtherCAT.Term_9_EK1100.Term_10_EK1122.Term_23_EK1100.Term_31_EL3773.L3_Voltage_Status.U3_Status/Error <-> L3 Voltage Status/U3 Status/Error
//     PlcTask Inputs/GVL_iXlinker.Device_2_EtherCAT.Term_9_EK1100.Term_10_EK1122.Term_23_EK1100.Term_31_EL3773.L1_Voltage_Status.U1_Status/Limit_x <-> L1 Voltage Status/U1 Status/Limit
//     PlcTask Inputs/GVL_iXlinker.Device_2_EtherCAT.Term_9_EK1100.Term_10_EK1122.Term_23_EK1100.Term_31_EL3773.L2_Voltage_Status.U2_Status/Limit_x <-> L2 Voltage Status/U2 Status/Limit
//     PlcTask Inputs/GVL_iXlinker.Device_2_EtherCAT.Term_9_EK1100.Term_10_EK1122.Term_23_EK1100.Term_31_EL3773.L3_Voltage_Status.U3_Status/Limit_x <-> L3 Voltage Status/U3 Status/Limit
//     PlcTask Inputs/GVL_iXlinker.Device_2_EtherCAT.Term_9_EK1100.Term_10_EK1122.Term_23_EK1100.Term_31_EL3773.L1_Voltage_Status.U1_Status/Overrange <-> L1 Voltage Status/U1 Status/Overrange
//     PlcTask Inputs/GVL_iXlinker.Device_2_EtherCAT.Term_9_EK1100.Term_10_EK1122.Term_23_EK1100.Term_31_EL3773.L2_Voltage_Status.U2_Status/Overrange <-> L2 Voltage Status/U2 Status/Overrange
//     PlcTask Inputs/GVL_iXlinker.Device_2_EtherCAT.Term_9_EK1100.Term_10_EK1122.Term_23_EK1100.Term_31_EL3773.L3_Voltage_Status.U3_Status/Overrange <-> L3 Voltage Status/U3 Status/Overrange
//     PlcTask Inputs/GVL_iXlinker.Device_2_EtherCAT.Term_9_EK1100.Term_10_EK1122.Term_23_EK1100.Term_31_EL3773.L1_Voltage_Status.U1_Status/Sync_error <-> L1 Voltage Status/U1 Status/Sync error
//     PlcTask Inputs/GVL_iXlinker.Device_2_EtherCAT.Term_9_EK1100.Term_10_EK1122.Term_23_EK1100.Term_31_EL3773.L2_Voltage_Status.U2_Status/Sync_error <-> L2 Voltage Status/U2 Status/Sync error
//     PlcTask Inputs/GVL_iXlinker.Device_2_EtherCAT.Term_9_EK1100.Term_10_EK1122.Term_23_EK1100.Term_31_EL3773.L3_Voltage_Status.U3_Status/Sync_error <-> L3 Voltage Status/U3 Status/Sync error
//     PlcTask Inputs/GVL_iXlinker.Device_2_EtherCAT.Term_9_EK1100.Term_10_EK1122.Term_23_EK1100.Term_31_EL3773.L1_Voltage_Status.U1_Status/TxPDO_State <-> L1 Voltage Status/U1 Status/TxPDO State
//     PlcTask Inputs/GVL_iXlinker.Device_2_EtherCAT.Term_9_EK1100.Term_10_EK1122.Term_23_EK1100.Term_31_EL3773.L2_Voltage_Status.U2_Status/TxPDO_State <-> L2 Voltage Status/U2 Status/TxPDO State
//     PlcTask Inputs/GVL_iXlinker.Device_2_EtherCAT.Term_9_EK1100.Term_10_EK1122.Term_23_EK1100.Term_31_EL3773.L3_Voltage_Status.U3_Status/TxPDO_State <-> L3 Voltage Status/U3 Status/TxPDO State
//     PlcTask Inputs/GVL_iXlinker.Device_2_EtherCAT.Term_9_EK1100.Term_10_EK1122.Term_23_EK1100.Term_31_EL3773.L1_Voltage_Status.U1_Status/TxPDO_Toggle <-> L1 Voltage Status/U1 Status/TxPDO Toggle
//     PlcTask Inputs/GVL_iXlinker.Device_2_EtherCAT.Term_9_EK1100.Term_10_EK1122.Term_23_EK1100.Term_31_EL3773.L2_Voltage_Status.U2_Status/TxPDO_Toggle <-> L2 Voltage Status/U2 Status/TxPDO Toggle
//     PlcTask Inputs/GVL_iXlinker.Device_2_EtherCAT.Term_9_EK1100.Term_10_EK1122.Term_23_EK1100.Term_31_EL3773.L3_Voltage_Status.U3_Status/TxPDO_Toggle <-> L3 Voltage Status/U3 Status/TxPDO Toggle
//     PlcTask Inputs/GVL_iXlinker.Device_2_EtherCAT.Term_9_EK1100.Term_10_EK1122.Term_23_EK1100.Term_31_EL3773.L1_Voltage_Status.U1_Status/Underrange <-> L1 Voltage Status/U1 Status/Underrange
//     PlcTask Inputs/GVL_iXlinker.Device_2_EtherCAT.Term_9_EK1100.Term_10_EK1122.Term_23_EK1100.Term_31_EL3773.L2_Voltage_Status.U2_Status/Underrange <-> L2 Voltage Status/U2 Status/Underrange
//     PlcTask Inputs/GVL_iXlinker.Device_2_EtherCAT.Term_9_EK1100.Term_10_EK1122.Term_23_EK1100.Term_31_EL3773.L3_Voltage_Status.U3_Status/Underrange <-> L3 Voltage Status/U3 Status/Underrange
//     PlcTask Inputs/GVL_iXlinker.Device_2_EtherCAT.Term_9_EK1100.Term_10_EK1122.Term_23_EK1100.Term_31_EL3773.WcState.InputToggle <-> WcState/InputToggle
//     PlcTask Inputs/GVL_iXlinker.Device_2_EtherCAT.Term_9_EK1100.Term_10_EK1122.Term_23_EK1100.Term_31_EL3773.WcState.WcState <-> WcState/WcState
//   Plc1/Plc1 Instance <-> Device 2 (EtherCAT)/Term 9 (EK1100)/Term 10 (EK1122)/Term 23 (EK1100)/Term 32 (EL2258)
//     PlcTask Inputs/GVL_iXlinker.Device_2_EtherCAT.Term_9_EK1100.Term_10_EK1122.Term_23_EK1100.Term_32_EL2258.InfoData.AdsAddr <-> InfoData/AdsAddr
//     PlcTask Inputs/GVL_iXlinker.Device_2_EtherCAT.Term_9_EK1100.Term_10_EK1122.Term_23_EK1100.Term_32_EL2258.InfoData.DcInputShift <-> InfoData/DcInputShift
//     PlcTask Inputs/GVL_iXlinker.Device_2_EtherCAT.Term_9_EK1100.Term_10_EK1122.Term_23_EK1100.Term_32_EL2258.InfoData.DcOutputShift <-> InfoData/DcOutputShift
//     PlcTask Inputs/GVL_iXlinker.Device_2_EtherCAT.Term_9_EK1100.Term_10_EK1122.Term_23_EK1100.Term_32_EL2258.InfoData.State <-> InfoData/State
//     PlcTask Inputs/GVL_iXlinker.Device_2_EtherCAT.Term_9_EK1100.Term_10_EK1122.Term_23_EK1100.Term_32_EL2258.MTO_Inputs_Channel_{1..8}.Status/Events_in_output_buffer <-> MTO Inputs Channel {1..8}/Status/Events in output buffer  (8 links)
//     PlcTask Inputs/GVL_iXlinker.Device_2_EtherCAT.Term_9_EK1100.Term_10_EK1122.Term_23_EK1100.Term_32_EL2258.MTO_Inputs_Channel_{1..8}.Status/Input_cycle_counter <-> MTO Inputs Channel {1..8}/Status/Input cycle counter  (8 links)
//     PlcTask Inputs/GVL_iXlinker.Device_2_EtherCAT.Term_9_EK1100.Term_10_EK1122.Term_23_EK1100.Term_32_EL2258.MTO_Inputs_Channel_{1..8}.Status/Output_buffer_overflow <-> MTO Inputs Channel {1..8}/Status/Output buffer overflow  (8 links)
//     PlcTask Inputs/GVL_iXlinker.Device_2_EtherCAT.Term_9_EK1100.Term_10_EK1122.Term_23_EK1100.Term_32_EL2258.MTO_Inputs_Channel_{1..8}.Status/Output_order_feedback <-> MTO Inputs Channel {1..8}/Status/Output order feedback  (8 links)
//     PlcTask Inputs/GVL_iXlinker.Device_2_EtherCAT.Term_9_EK1100.Term_10_EK1122.Term_23_EK1100.Term_32_EL2258.MTO_Inputs_Channel_{1..8}.Status/Output_short_circuit <-> MTO Inputs Channel {1..8}/Status/Output short circuit  (8 links)
//     PlcTask Inputs/GVL_iXlinker.Device_2_EtherCAT.Term_9_EK1100.Term_10_EK1122.Term_23_EK1100.Term_32_EL2258.MTO_Inputs_Channel_{1..8}.Status/Output_state <-> MTO Inputs Channel {1..8}/Status/Output state  (8 links)
//     PlcTask Inputs/GVL_iXlinker.Device_2_EtherCAT.Term_9_EK1100.Term_10_EK1122.Term_23_EK1100.Term_32_EL2258.WcState.InputToggle <-> WcState/InputToggle
//     PlcTask Inputs/GVL_iXlinker.Device_2_EtherCAT.Term_9_EK1100.Term_10_EK1122.Term_23_EK1100.Term_32_EL2258.WcState.WcState <-> WcState/WcState
//     PlcTask Outputs/GVL_iXlinker.Device_2_EtherCAT.Term_9_EK1100.Term_10_EK1122.Term_23_EK1100.Term_32_EL2258.MTO_Outputs_10x_Channel_{1..8}.Ctrl/Enable_manual_operation <-> MTO Outputs 10x Channel {1..8}/Ctrl/Enable manual operation  (8 links)
//     PlcTask Outputs/GVL_iXlinker.Device_2_EtherCAT.Term_9_EK1100.Term_10_EK1122.Term_23_EK1100.Term_32_EL2258.MTO_Outputs_10x_Channel_{1..8}.Ctrl/Force_order <-> MTO Outputs 10x Channel {1..8}/Ctrl/Force order  (8 links)
//     PlcTask Outputs/GVL_iXlinker.Device_2_EtherCAT.Term_9_EK1100.Term_10_EK1122.Term_23_EK1100.Term_32_EL2258.MTO_Outputs_10x_Channel_{1..8}.Ctrl/Manual_output_state <-> MTO Outputs 10x Channel {1..8}/Ctrl/Manual output state  (8 links)
//     PlcTask Outputs/GVL_iXlinker.Device_2_EtherCAT.Term_9_EK1100.Term_10_EK1122.Term_23_EK1100.Term_32_EL2258.MTO_Outputs_10x_Channel_{1..8}.Ctrl/No_of_output_events <-> MTO Outputs 10x Channel {1..8}/Ctrl/No of output events  (8 links)
//     PlcTask Outputs/GVL_iXlinker.Device_2_EtherCAT.Term_9_EK1100.Term_10_EK1122.Term_23_EK1100.Term_32_EL2258.MTO_Outputs_10x_Channel_{1..8}.Ctrl/Output_buffer_reset <-> MTO Outputs 10x Channel {1..8}/Ctrl/Output buffer reset  (8 links)
//     PlcTask Outputs/GVL_iXlinker.Device_2_EtherCAT.Term_9_EK1100.Term_10_EK1122.Term_23_EK1100.Term_32_EL2258.MTO_Outputs_10x_Channel_{1..8}.Ctrl/Output_order_counter <-> MTO Outputs 10x Channel {1..8}/Ctrl/Output order counter  (8 links)
//     PlcTask Outputs/GVL_iXlinker.Device_2_EtherCAT.Term_9_EK1100.Term_10_EK1122.Term_23_EK1100.Term_32_EL2258.MTO_Outputs_10x_Channel_1.Output_event_time[0] <-> MTO Outputs 10x Channel 1/Output event time 1
//     PlcTask Outputs/GVL_iXlinker.Device_2_EtherCAT.Term_9_EK1100.Term_10_EK1122.Term_23_EK1100.Term_32_EL2258.MTO_Outputs_10x_Channel_1.Output_event_time[1] <-> MTO Outputs 10x Channel 1/Output event time 2
//     PlcTask Outputs/GVL_iXlinker.Device_2_EtherCAT.Term_9_EK1100.Term_10_EK1122.Term_23_EK1100.Term_32_EL2258.MTO_Outputs_10x_Channel_1.Output_event_time[2] <-> MTO Outputs 10x Channel 1/Output event time 3
//     PlcTask Outputs/GVL_iXlinker.Device_2_EtherCAT.Term_9_EK1100.Term_10_EK1122.Term_23_EK1100.Term_32_EL2258.MTO_Outputs_10x_Channel_1.Output_event_time[3] <-> MTO Outputs 10x Channel 1/Output event time 4
//     PlcTask Outputs/GVL_iXlinker.Device_2_EtherCAT.Term_9_EK1100.Term_10_EK1122.Term_23_EK1100.Term_32_EL2258.MTO_Outputs_10x_Channel_1.Output_event_time[4] <-> MTO Outputs 10x Channel 1/Output event time 5
//     PlcTask Outputs/GVL_iXlinker.Device_2_EtherCAT.Term_9_EK1100.Term_10_EK1122.Term_23_EK1100.Term_32_EL2258.MTO_Outputs_10x_Channel_1.Output_event_time[5] <-> MTO Outputs 10x Channel 1/Output event time 6
//     PlcTask Outputs/GVL_iXlinker.Device_2_EtherCAT.Term_9_EK1100.Term_10_EK1122.Term_23_EK1100.Term_32_EL2258.MTO_Outputs_10x_Channel_1.Output_event_time[6] <-> MTO Outputs 10x Channel 1/Output event time 7
//     PlcTask Outputs/GVL_iXlinker.Device_2_EtherCAT.Term_9_EK1100.Term_10_EK1122.Term_23_EK1100.Term_32_EL2258.MTO_Outputs_10x_Channel_1.Output_event_time[7] <-> MTO Outputs 10x Channel 1/Output event time 8
//     PlcTask Outputs/GVL_iXlinker.Device_2_EtherCAT.Term_9_EK1100.Term_10_EK1122.Term_23_EK1100.Term_32_EL2258.MTO_Outputs_10x_Channel_1.Output_event_time[8] <-> MTO Outputs 10x Channel 1/Output event time 9
//     PlcTask Outputs/GVL_iXlinker.Device_2_EtherCAT.Term_9_EK1100.Term_10_EK1122.Term_23_EK1100.Term_32_EL2258.MTO_Outputs_10x_Channel_1.Output_event_time[9] <-> MTO Outputs 10x Channel 1/Output event time 10
//     PlcTask Outputs/GVL_iXlinker.Device_2_EtherCAT.Term_9_EK1100.Term_10_EK1122.Term_23_EK1100.Term_32_EL2258.MTO_Outputs_10x_Channel_2.Output_event_time[0] <-> MTO Outputs 10x Channel 2/Output event time 1
//     PlcTask Outputs/GVL_iXlinker.Device_2_EtherCAT.Term_9_EK1100.Term_10_EK1122.Term_23_EK1100.Term_32_EL2258.MTO_Outputs_10x_Channel_2.Output_event_time[1] <-> MTO Outputs 10x Channel 2/Output event time 2
//     PlcTask Outputs/GVL_iXlinker.Device_2_EtherCAT.Term_9_EK1100.Term_10_EK1122.Term_23_EK1100.Term_32_EL2258.MTO_Outputs_10x_Channel_2.Output_event_time[2] <-> MTO Outputs 10x Channel 2/Output event time 3
//     PlcTask Outputs/GVL_iXlinker.Device_2_EtherCAT.Term_9_EK1100.Term_10_EK1122.Term_23_EK1100.Term_32_EL2258.MTO_Outputs_10x_Channel_2.Output_event_time[3] <-> MTO Outputs 10x Channel 2/Output event time 4
//     PlcTask Outputs/GVL_iXlinker.Device_2_EtherCAT.Term_9_EK1100.Term_10_EK1122.Term_23_EK1100.Term_32_EL2258.MTO_Outputs_10x_Channel_2.Output_event_time[4] <-> MTO Outputs 10x Channel 2/Output event time 5
//     PlcTask Outputs/GVL_iXlinker.Device_2_EtherCAT.Term_9_EK1100.Term_10_EK1122.Term_23_EK1100.Term_32_EL2258.MTO_Outputs_10x_Channel_2.Output_event_time[5] <-> MTO Outputs 10x Channel 2/Output event time 6
//     PlcTask Outputs/GVL_iXlinker.Device_2_EtherCAT.Term_9_EK1100.Term_10_EK1122.Term_23_EK1100.Term_32_EL2258.MTO_Outputs_10x_Channel_2.Output_event_time[6] <-> MTO Outputs 10x Channel 2/Output event time 7
//     PlcTask Outputs/GVL_iXlinker.Device_2_EtherCAT.Term_9_EK1100.Term_10_EK1122.Term_23_EK1100.Term_32_EL2258.MTO_Outputs_10x_Channel_2.Output_event_time[7] <-> MTO Outputs 10x Channel 2/Output event time 8
//     PlcTask Outputs/GVL_iXlinker.Device_2_EtherCAT.Term_9_EK1100.Term_10_EK1122.Term_23_EK1100.Term_32_EL2258.MTO_Outputs_10x_Channel_2.Output_event_time[8] <-> MTO Outputs 10x Channel 2/Output event time 9
//     PlcTask Outputs/GVL_iXlinker.Device_2_EtherCAT.Term_9_EK1100.Term_10_EK1122.Term_23_EK1100.Term_32_EL2258.MTO_Outputs_10x_Channel_2.Output_event_time[9] <-> MTO Outputs 10x Channel 2/Output event time 10
//     PlcTask Outputs/GVL_iXlinker.Device_2_EtherCAT.Term_9_EK1100.Term_10_EK1122.Term_23_EK1100.Term_32_EL2258.MTO_Outputs_10x_Channel_3.Output_event_time[0] <-> MTO Outputs 10x Channel 3/Output event time 1
//     PlcTask Outputs/GVL_iXlinker.Device_2_EtherCAT.Term_9_EK1100.Term_10_EK1122.Term_23_EK1100.Term_32_EL2258.MTO_Outputs_10x_Channel_3.Output_event_time[1] <-> MTO Outputs 10x Channel 3/Output event time 2
//     PlcTask Outputs/GVL_iXlinker.Device_2_EtherCAT.Term_9_EK1100.Term_10_EK1122.Term_23_EK1100.Term_32_EL2258.MTO_Outputs_10x_Channel_3.Output_event_time[2] <-> MTO Outputs 10x Channel 3/Output event time 3
//     PlcTask Outputs/GVL_iXlinker.Device_2_EtherCAT.Term_9_EK1100.Term_10_EK1122.Term_23_EK1100.Term_32_EL2258.MTO_Outputs_10x_Channel_3.Output_event_time[3] <-> MTO Outputs 10x Channel 3/Output event time 4
//     PlcTask Outputs/GVL_iXlinker.Device_2_EtherCAT.Term_9_EK1100.Term_10_EK1122.Term_23_EK1100.Term_32_EL2258.MTO_Outputs_10x_Channel_3.Output_event_time[4] <-> MTO Outputs 10x Channel 3/Output event time 5
//     PlcTask Outputs/GVL_iXlinker.Device_2_EtherCAT.Term_9_EK1100.Term_10_EK1122.Term_23_EK1100.Term_32_EL2258.MTO_Outputs_10x_Channel_3.Output_event_time[5] <-> MTO Outputs 10x Channel 3/Output event time 6
//     PlcTask Outputs/GVL_iXlinker.Device_2_EtherCAT.Term_9_EK1100.Term_10_EK1122.Term_23_EK1100.Term_32_EL2258.MTO_Outputs_10x_Channel_3.Output_event_time[6] <-> MTO Outputs 10x Channel 3/Output event time 7
//     PlcTask Outputs/GVL_iXlinker.Device_2_EtherCAT.Term_9_EK1100.Term_10_EK1122.Term_23_EK1100.Term_32_EL2258.MTO_Outputs_10x_Channel_3.Output_event_time[7] <-> MTO Outputs 10x Channel 3/Output event time 8
//     PlcTask Outputs/GVL_iXlinker.Device_2_EtherCAT.Term_9_EK1100.Term_10_EK1122.Term_23_EK1100.Term_32_EL2258.MTO_Outputs_10x_Channel_3.Output_event_time[8] <-> MTO Outputs 10x Channel 3/Output event time 9
//     PlcTask Outputs/GVL_iXlinker.Device_2_EtherCAT.Term_9_EK1100.Term_10_EK1122.Term_23_EK1100.Term_32_EL2258.MTO_Outputs_10x_Channel_3.Output_event_time[9] <-> MTO Outputs 10x Channel 3/Output event time 10
//     PlcTask Outputs/GVL_iXlinker.Device_2_EtherCAT.Term_9_EK1100.Term_10_EK1122.Term_23_EK1100.Term_32_EL2258.MTO_Outputs_10x_Channel_4.Output_event_time[0] <-> MTO Outputs 10x Channel 4/Output event time 1
//     PlcTask Outputs/GVL_iXlinker.Device_2_EtherCAT.Term_9_EK1100.Term_10_EK1122.Term_23_EK1100.Term_32_EL2258.MTO_Outputs_10x_Channel_4.Output_event_time[1] <-> MTO Outputs 10x Channel 4/Output event time 2
//     PlcTask Outputs/GVL_iXlinker.Device_2_EtherCAT.Term_9_EK1100.Term_10_EK1122.Term_23_EK1100.Term_32_EL2258.MTO_Outputs_10x_Channel_4.Output_event_time[2] <-> MTO Outputs 10x Channel 4/Output event time 3
//     PlcTask Outputs/GVL_iXlinker.Device_2_EtherCAT.Term_9_EK1100.Term_10_EK1122.Term_23_EK1100.Term_32_EL2258.MTO_Outputs_10x_Channel_4.Output_event_time[3] <-> MTO Outputs 10x Channel 4/Output event time 4
//     PlcTask Outputs/GVL_iXlinker.Device_2_EtherCAT.Term_9_EK1100.Term_10_EK1122.Term_23_EK1100.Term_32_EL2258.MTO_Outputs_10x_Channel_4.Output_event_time[4] <-> MTO Outputs 10x Channel 4/Output event time 5
//     PlcTask Outputs/GVL_iXlinker.Device_2_EtherCAT.Term_9_EK1100.Term_10_EK1122.Term_23_EK1100.Term_32_EL2258.MTO_Outputs_10x_Channel_4.Output_event_time[5] <-> MTO Outputs 10x Channel 4/Output event time 6
//     PlcTask Outputs/GVL_iXlinker.Device_2_EtherCAT.Term_9_EK1100.Term_10_EK1122.Term_23_EK1100.Term_32_EL2258.MTO_Outputs_10x_Channel_4.Output_event_time[6] <-> MTO Outputs 10x Channel 4/Output event time 7
//     PlcTask Outputs/GVL_iXlinker.Device_2_EtherCAT.Term_9_EK1100.Term_10_EK1122.Term_23_EK1100.Term_32_EL2258.MTO_Outputs_10x_Channel_4.Output_event_time[7] <-> MTO Outputs 10x Channel 4/Output event time 8
//     PlcTask Outputs/GVL_iXlinker.Device_2_EtherCAT.Term_9_EK1100.Term_10_EK1122.Term_23_EK1100.Term_32_EL2258.MTO_Outputs_10x_Channel_4.Output_event_time[8] <-> MTO Outputs 10x Channel 4/Output event time 9
//     PlcTask Outputs/GVL_iXlinker.Device_2_EtherCAT.Term_9_EK1100.Term_10_EK1122.Term_23_EK1100.Term_32_EL2258.MTO_Outputs_10x_Channel_4.Output_event_time[9] <-> MTO Outputs 10x Channel 4/Output event time 10
//     PlcTask Outputs/GVL_iXlinker.Device_2_EtherCAT.Term_9_EK1100.Term_10_EK1122.Term_23_EK1100.Term_32_EL2258.MTO_Outputs_10x_Channel_5.Output_event_time[0] <-> MTO Outputs 10x Channel 5/Output event time 1
//     PlcTask Outputs/GVL_iXlinker.Device_2_EtherCAT.Term_9_EK1100.Term_10_EK1122.Term_23_EK1100.Term_32_EL2258.MTO_Outputs_10x_Channel_5.Output_event_time[1] <-> MTO Outputs 10x Channel 5/Output event time 2
//     PlcTask Outputs/GVL_iXlinker.Device_2_EtherCAT.Term_9_EK1100.Term_10_EK1122.Term_23_EK1100.Term_32_EL2258.MTO_Outputs_10x_Channel_5.Output_event_time[2] <-> MTO Outputs 10x Channel 5/Output event time 3
//     PlcTask Outputs/GVL_iXlinker.Device_2_EtherCAT.Term_9_EK1100.Term_10_EK1122.Term_23_EK1100.Term_32_EL2258.MTO_Outputs_10x_Channel_5.Output_event_time[3] <-> MTO Outputs 10x Channel 5/Output event time 4
//     PlcTask Outputs/GVL_iXlinker.Device_2_EtherCAT.Term_9_EK1100.Term_10_EK1122.Term_23_EK1100.Term_32_EL2258.MTO_Outputs_10x_Channel_5.Output_event_time[4] <-> MTO Outputs 10x Channel 5/Output event time 5
//     PlcTask Outputs/GVL_iXlinker.Device_2_EtherCAT.Term_9_EK1100.Term_10_EK1122.Term_23_EK1100.Term_32_EL2258.MTO_Outputs_10x_Channel_5.Output_event_time[5] <-> MTO Outputs 10x Channel 5/Output event time 6
//     PlcTask Outputs/GVL_iXlinker.Device_2_EtherCAT.Term_9_EK1100.Term_10_EK1122.Term_23_EK1100.Term_32_EL2258.MTO_Outputs_10x_Channel_5.Output_event_time[6] <-> MTO Outputs 10x Channel 5/Output event time 7
//     PlcTask Outputs/GVL_iXlinker.Device_2_EtherCAT.Term_9_EK1100.Term_10_EK1122.Term_23_EK1100.Term_32_EL2258.MTO_Outputs_10x_Channel_5.Output_event_time[7] <-> MTO Outputs 10x Channel 5/Output event time 8
//     PlcTask Outputs/GVL_iXlinker.Device_2_EtherCAT.Term_9_EK1100.Term_10_EK1122.Term_23_EK1100.Term_32_EL2258.MTO_Outputs_10x_Channel_5.Output_event_time[8] <-> MTO Outputs 10x Channel 5/Output event time 9
//     PlcTask Outputs/GVL_iXlinker.Device_2_EtherCAT.Term_9_EK1100.Term_10_EK1122.Term_23_EK1100.Term_32_EL2258.MTO_Outputs_10x_Channel_5.Output_event_time[9] <-> MTO Outputs 10x Channel 5/Output event time 10
//     PlcTask Outputs/GVL_iXlinker.Device_2_EtherCAT.Term_9_EK1100.Term_10_EK1122.Term_23_EK1100.Term_32_EL2258.MTO_Outputs_10x_Channel_6.Output_event_time[0] <-> MTO Outputs 10x Channel 6/Output event time 1
